(* IEC 61131-3 sources: Nauka-PLC-ST/, 81 files *)

(* ---- Zaawansowany_sterownik_prasy_hydraulicznej.st ---- *)
VAR
  stanAktualny               : stanPrasy;
  Przycisk_1                 : BOOL;  // pierwszy reczny przycisk uruchamiajacy prace ukladu
  Przycisk_2                 : BOOL;  // drugi reczny przycisk uruchamiajacy prace ukladu
  Dolna_krancowka_silownika  : BOOL;  // przelacznik krancowy wykrywajacy wysuniecie silownika
  Gorna_krancowka_silownika  : BOOL;  // przelacznik krancowy wykrywajacy wsuniecie silownika
  Timer_prasowanie           : TON;   // czas prasowania detalu
  Zawor_A                    : BOOL;  // zawor wysuwajacy prase w dol
  Zawor_B                    : BOOL;  // zawor wsuwajacy prase do gory
END_VAR

Timer_prasowanie(IN := Dolna_krancowka, PT := T#3S)

TYPE stanPrasy :
(
  OCZEKIWANIE
  RUCH_W_DOL
  PRASOWANIE
  RUCH_W_GORE
  ALARM
);
END_TYPE

CASE stanAktualny OF
    OCZEKIWANIE:
        Zawor_A := FALSE;
        Zawor_B := TRUE; // prasa czeka w górze

        // Warunek startu: Oba przyciski
        IF Przycisk_1 AND Przycisk_2 THEN
            stanAktualny := RUCH_W_DOL;
        END_IF;

    RUCH_W_DOL:
        Zawor_A := TRUE;  // Jedziemy w dół
        Zawor_B := FALSE;

        // oczekiwanie na stan wysoki od dolnej krancowki
        IF Dolna_krancowka_silownika THEN
            stanAktualny := PRASOWANIE;
        END_IF;

    PRASOWANIE:
        // wlaczamy timer (IN := TRUE)
        Timer_prasowanie(IN := TRUE, PT := T#3S);

        IF Timer_prasowanie.Q THEN
            Timer_prasowanie(IN := FALSE); // reset timera przed powrotem
            stanAktualny := RUCH_W_GORE;
        END_IF;

    RUCH_W_GORE:
        Zawor_A := FALSE;
        Zawor_B := TRUE; // powrot prasy do stanu poczatkowego

        IF Gorna_krancowka_silownika THEN
            stanAktualny := OCZEKIWANIE;
        END_IF;

    ALARM:
        Zawor_A := FALSE;
        Zawor_B := FALSE; // sytuacja awaryjna
END_CASE

(* ---- Motor_Control_Diagnostic.st ---- *)
FUNCTION_BLOCK Motor_control_diagnostic
VAR_INPUT
    xStart    : BOOL; // Przycisk Start
    xStop     : BOOL; // Przycisk Stop
    xFeedback : BOOL; // Potwierdzenie, ze silnik faktycznie ruszyl
    xErrorIn  : BOOL; // Awaria zewnetrzna (np. termik)
    xReset    : BOOL; // Przycisk do kasowania bledu
END_VAR

VAR_OUTPUT
    xRun      : BOOL;   // Wyjscie na stycznik silnika
    xAlarm    : BOOL;   // Lampka alarmu
    sStatus   : STRING; // Tekstowy opis na ekran HMI
END_VAR

VAR
    Timer_Potw : TON; // Zegar/czasowka
END_VAR

// --- 1. LOGIKA START / STOP ---
// Silnik rusza, gdy wciskasz Start, pod warunkiem, ze nie ma awarii i alarmu
IF xStart AND NOT xErrorIn AND NOT xAlarm THEN
    xRun := TRUE;
    sStatus := 'Silnik pracuje';
END_IF;

// Silnik staje, gdy: wcisniesz Stop, wywali blad (ErrorIn) lub pojawi sie Alarm
IF xStop OR xErrorIn OR xAlarm THEN
    xRun := FALSE;
    // Jesli to nie byl alarm, ustaw status na postoj
    IF NOT xAlarm THEN
        sStatus := 'Postoj';
    END_IF;
END_IF;

// --- 2. CZASOWKA (DIAGNOSTYKA) ---
// Timer liczy, gdy: wykonuje sie praca (xRun), ale nie widzisz potwierdzenia (NOT xFeedback)
Timer_Potw(IN := (xRun AND NOT xFeedback), PT := T#2s);

// --- 3. REAKCJA NA BLAD ---
// Jesli timer doliczyl do 2 sekund (Q), to znaczy, ze cos jest nie tak
IF Timer_Potw.Q THEN
    xAlarm  := TRUE;             // Wlaczamy alarm
    sStatus := 'Blad potwierdzenia'; // Opisujemy blad
    xRun    := FALSE;            // Wylaczamy silnik dla bezpieczenstwa
END_IF;

// --- 4. KASOWANIE ALARMU ---
// Gdy operator wcisnie Reset, czyscimy alarm i status
IF xReset THEN
    xAlarm := FALSE;
    sStatus := 'Gotowy';
END_IF;

(* ---- Obsluga_alarmow_analogowych.st ---- *)
FUNCTION_BLOCK Obsluga_alarmow_analogowych

VAR_INPUT
    Wartosc_Skalowana : REAL;    // Wartosc przeliczona
    Prog_Wysoki       : REAL;    // Prog alarmu
    Prog_Krytyczny    : REAL;    // Prog krytycznej wartosci w ukladzie
    Histereza         : REAL := 1.0; // Zapobiega przeciwko tzw drganiu stykow
END_VAR

VAR_OUTPUT
    Ostrzezenie : BOOL; // Informacja o przekroczeniu progu wysokiego
    Alarm       : BOOL; // Informacja o przekroczeniu progu krytycznego
END_VAR

// 1. Sprawdzenie progu krytycznego - natychmiastowe zatrzymanie, gdy zostanie przekroczona wartosc krytyczna
IF Wartosc_Skalowana >= Prog_Krytyczny THEN
    Alarm := TRUE;  // Informacja o przekroczeniu progu krytycznego
ELSIF Wartosc_Skalowana <= (Prog_Krytyczny - Histereza) THEN  // Wylacz alarm po powrocie do bezpiecznej wartosci
    Alarm := FALSE;  // Wylacz alarm
END_IF;

// 2. Ostrzezenie - tylko sygnalizacja
IF Wartosc_Skalowana >= Prog_Wysoki THEN
    Ostrzezenie := TRUE;  // Sygnalizacja przekroczenia normy np. lampka
ELSIF Wartosc_Skalowana <= (Prog_Wysoki - Histereza) THEN // Wylacz jesli spadnie ponizej tego progu
    Ostrzezenie := FALSE;
END_IF;

(* ---- Skalowanie_Analogowe.st ---- *)
FUNCTION_BLOCK Skalowanie_Analogow
VAR_INPUT
    Sygnal_RAW      : INT;    // Faktyczny odczyt z karty
    Zakres_Wej_Min   : REAL := 0.0;
    Zakres_Wej_Max   : REAL := 27648.0;
    Limit_Dolny     : REAL := 0.0;     // np. 0 bar
    Limit_Gorny     : REAL := 100.0;   // np. 10 bar
END_VAR

VAR_OUTPUT
    Wynik_Skalowania : REAL;    // Wartość przeliczona
    Awaria_Czujnika  : BOOL;    // Błąd zakresu / przerwany przewod
END_VAR

VAR
    Pomoc_Real       : REAL;    // Przejście na wartosc przecinkowa
END_VAR

// 1. Przepisanie wartosci z czujnika na wartosc z przecinkiem
Pomoc_Real := INT_TO_REAL(Sygnal_RAW);

// 2. Skalowanie wartosci z czujnika na wartosci fizyczne
IF (Zakres_Wej_Max - Zakres_Wej_Min) <> 0 THEN
    Wynik_Skalowania := Limit_Dolny + (Pomoc_Real - Zakres_Wej_Min) * (Limit_Gorny - Limit_Dolny) / (Zakres_Wej_Max - Zakres_Wej_Min);
ELSE
    Wynik_Skalowania := 0.0;
    Awaria_Czujnika := TRUE;
END_IF;

// 3. Diagnostyka na wypadek awarii
IF Pomoc_Real < -500.0 OR Pomoc_Real > 30000.0 THEN
    Awaria_Czujnika := TRUE;
ELSE
    Awaria_Czujnika := FALSE;
END_IF;

(* ---- Automat_segregujacy.st ---- *)
VAR
    Krok : INT := 0;              // krok programu
    Start_Maszyny : BOOL;         // przycisk NO wlaczajacy maszyne
    E_Stop : BOOL;                // przycisk bezpieczeństwa NC

    Tasma : BOOL;                 // napęd taśmociągu
    Spychacz_Metal : BOOL;        // aiłownik zrzucający metal
    Spychacz_Plastik : BOOL;      // aiłownik zrzucający plastik

    Fotokomorka_wlotowa : BOOL;   // wykrycie obiektu na wejściu
    Czujnik_indukcyjny : BOOL;    // detekcja metalu
    Czujnik_pojemnosciowy : BOOL; // detekcja plastiku
    Krancowka_baza : BOOL;        // czujnik potwierdzajacy powrotu siłowników na pozycję startowa

    Timer_Dojazdu : TON;          // Odmierzenie drogi od czujnika do spychacza
END_VAR

// system bezpieczenstwa
IF NOT E_stop THEN
    Tasma := FALSE;
    Spychacz_metal := FALSE;
    Spychacz_plastik := FALSE;
    Krok := 0;
    RETURN;
END_IF;

Timer_Dojazdu(IN := (Krok = 20 OR Krok = 30), PT := T#3s);

CASE Krok OF
    0:  // IDLE: oczekiwanie na gotowosc systemu
        Tasma := FALSE;
        IF Start_maszyny THEN
            Krok := 10;
        END_IF;

    10: // taśma rusza i czeka na materiał
        Tasma := TRUE;
        IF Czujnik_indukcyjny THEN
            Krok := 20; // wykrycie metalu
        ELSIF Czujnik_pojemnosciowy THEN
            Krok := 30; // wykrycie plastiku
        END_IF;

    20: // transportowaie metalu do spychacza
        IF Timer_dojazdu.Q THEN
            Tasma := FALSE;
            Krok := 21;
        END_IF;

    21: // uzycie silownika
        Spychacz_metal := TRUE;
        IF NOT Krancowka_baza THEN  // wysuniety spychacz
            Krok := 22;
        END_IF;

    22: // powrot spychacza do bazy
        Spychacz_metal := FALSE;
        IF Krancowka_baza THEN
            Krok := 10; // oczekiwanie na kolejen smieci
        END_IF;

    30: // transport plastiku
        IF Timer_dojazdu.Q THEN
            Tasma := FALSE;
            Krok := 31;
        END_IF;

    31: // zrzut plastiku do pojemnika
        Spychacz_plastik := TRUE;
        IF NOT Krancowka_baza THEN
            Krok := 32;
        END_IF;

    32: // powrot do stanu wyjsciowego
        Spychacz_plastik := FALSE;
        IF Krancowka_baza THEN
            Krok := 10;
        END_IF;

END_CASE;

(* ---- Automatyczny_cykl_nawrotny.st ---- *)
VAR
    Stycznik_lewo  : BOOL;
    Stycznik_prawo : BOOL;
    Przycisk_start : BOOL;
    Przycisk_stop  : BOOL; // Zakladamy NC

    Timer_pracy    : TON;
    Timer_pauzy    : TON;

    Kierunek       : BOOL; // FALSE = Lewo, TRUE = Prawo
    Praca_aktywna  : BOOL; // Informuje o uruchomionym cyklu
END_VAR

// Start i Stop cyklu
IF Przycisk_start AND Przycisk_stop THEN
    Praca_aktywna := TRUE;
ELSIF NOT Przycisk_stop THEN
    Praca_aktywna := FALSE;
END_IF;

// Obsluga timerow
Timer_pracy(IN := Praca_aktywna AND NOT Timer_pauzy.IN, PT := T#5S);
Timer_pauzy(IN := Timer_pracy.Q, PT := T#3S); // Czas na wyhamowanie

// Zmiana kierunku po kazdej pauzie
IF Timer_pauzy.Q THEN
    Kierunek := NOT Kierunek; // Przelacz na przeciwny
END_IF;

// Kontrola stycznikow
Stycznik_lewo  := Praca_aktywna AND NOT Kierunek AND NOT Timer_pauzy.IN;
Stycznik_prawo := Praca_aktywna AND Kierunek AND NOT Timer_pauzy.IN;

(* ---- Automatyczny_mieszalnik.st ---- *)
// 1. Obsługa Stopu Awaryjnego (Reset wszystkiego)
IF NOT Stop_awaryjny THEN
    Krok_ukladu := 0;
    Zawor_A := FALSE;
    Zawor_B := FALSE;
    Mieszadlo := FALSE;
    Zawor_spustowy := FALSE;
END_IF;

// 2. Główna maszyna stanów
CASE Krok_ukladu OF
    0: // Oczekiwanie
        IF Start THEN
            Krok_ukladu := 10;
        END_IF;

    10: // Dolewanie A
        Zawor_A := TRUE;
        IF Czujnik_poziomu >= 40.0 THEN
            Zawor_A := FALSE; // Wyłączamy, gdy pełne!
            Krok_ukladu := 20;
        END_IF;

    20: // Dolewanie B
        Zawor_B := TRUE;
        IF Czujnik_poziomu >= 80.0 THEN // Używaj tej samej nazwy zmiennej poziomu
            Zawor_B := FALSE;
            Krok_ukladu := 30;
        END_IF;

    30: // Mieszanie
        Mieszadlo := TRUE;
        // Składnia timera: Czas_mieszania(IN := TRUE, PT := T#10S);
        IF Czas_mieszania.Q THEN
            Mieszadlo := FALSE;
            Krok_ukladu := 40;
        END_IF;

    40: // Opróżnianie
        Zawor_spustowy := TRUE;
        IF Czujnik_poziomu <= 2.0 THEN
            Zawor_spustowy := FALSE;
            Krok_ukladu := 0; // Koniec cyklu, wróć do początku
        END_IF;
END_CASE;

(* ---- Diagnostyka_uszkodzenia_czujnika.st ---- *)
VAR
  wartoscCzujnik : REAL;  // wartosc odczytana z czujnika
  ostatniaWartosc : REAL;  // ostatnia wartosc z czujnika
  timerKontrola : TON;  // czas sprawdzania wartosci zmiany
  bladCzujnika : BOOL;  // pamiec bledu
  tolercjaSygnalu : REAL := 0.01;  // minimalna mozliwa zmiana aby program ja zauwazyl
END_VAR

// sprawdzenie odleglosci miedzy dwiema liczbami
IF ABS(wartoscCzujnik - ostatniaWartosc) < tolercjaSygnalu THEN
    // gdy tolerancja miedzy sygnalami jest za mala to uruchom odliczanie
    timerKontrola.IN := TRUE;
ELSE
    // gdy jednak sygnal sie zmienia to zresetuj timer
    timerKontrola.IN := FALSE;
END_IF;

timerKontrola.PT := T#10s; // deadline ze czujnik jest uszkodzony
timerKontrola();           // wywolanie timera kontroli sygnalu

IF timerKontrola.Q THEN
    bladCzujnika := TRUE;  // sygnalizacja alarmu
END_IF;

ostatniaWartosc := wartoscCzujnik;  // zapamietanie ostatniej wartosci czujnika

(* ---- Emergency_Stop.st ---- *)
PROGRAM SafetyLogic
VAR
    // WEJŚCIA
    bEStop_NC    : BOOL;    // Przycisk bezpieczeństwa (Fizycznie NC - Normalnie Zamknięty)
    bReset_Button : BOOL;   // Przycisk Reset (NO)

    // WYJŚCIA
    bSafetyOK    : BOOL;    // Flaga bezpieczeństwa - zezwolenie na pracę
    bError_Lamp  : BOOL;    // Lampa błędu (miga, gdy brak bezpieczeństwa)
END_VAR

// 1. Logika bezpieczeństwa
// Jeśli grzyb jest wciśnięty (bEStop_NC = FALSE), bezpieczeństwo zostaje przerwane
IF NOT bEStop_NC THEN
    bSafetyOK := FALSE;
END_IF

// 2. Warunek Resetu
// Bezpieczeństwo można przywrócić tylko, gdy grzyb jest wyciągnięty (TRUE)
// i naciśniemy przycisk Reset
IF bEStop_NC AND bReset_Button THEN
    bSafetyOK := TRUE;
END_IF

// 3. Sygnalizacja
bError_Lamp := NOT bSafetyOK;

END_PROGRAM

(* ---- Inteligentny_garaz.st ---- *)
VAR
    Wylacznik_ukladu    : BOOL;  // przcycisk bistabilny NC wylaczajacy brame
    Pilot_bramy         : BOOL;  // przycisk monostabilny NO otwierajacy brame
    Czujnik_ruchu_1     : BOOL;  // czujnik ruchu nr 1 w okolicach bramy
    Czujnik_ruchu_2     : BOOL;  // czujnik ruchu nr 2 w okolicach bramy
    Przycisk_serwisowy  : BOOL;  // przycisk NO monostabilny wlaczajacy swiatło na stałe
    Czujnik_CO2         : BOOL;  // czujnik wykrywajacy CO2 w powietrzu
    Potwierdzenie_went  : BOOL;  // potwierdzenie pracy wentylatora

    // --- WYJŚCIA (Fizyczne) ---
    Silnik_bramy        : BOOL;  // umozliwia wjazd samochodu
    Oswietlenie_bramy   : BOOL;  // oswietlenie bramy garazowej
    Wentylator          : BOOL;  // urzadzenie z podtrzymaniem
    Alarm_CO2           : BOOL; // czerwona lampka
    Alarm_Awaria_Went   : BOOL; // bład wentylatora/awaria wentylatora

    // --- BLOKI CZASOWE ---
    Timer_swiatlo       : TOF; // podtrzymanie światla po ruchu
    Timer_wentylator    : TOF; // podtrzymuje wietrzenie po zniknieciu gazu
    Timer_awaria_went   : TON; // odliczanie czasu na potwierdzenie pracy
END_VAR

// swiatlo reaguje na ruch, pdtrzymuje 30s po zniknieciu ruchu
Timer_swiatlo(IN := (Czujnik_ruchu_1 OR Czujnik_ruchu_2), PT := T#30s);

// wentylacja reaguje na gaz, trzyma 10s po oczyszczeniu powietrza
Timer_wentylator(IN := Czujnik_CO2, PT := T#10s);

// diagnostyka jeśli wentylator ma pracowac, a nie ma potwierdzenia przez 5s, a musi byc potwierdzenie
Timer_awaria_went(IN := Wentylator AND NOT Potwierdzenie_went, PT := T#5s);

// brama otwiera się z pilota, o ile nie ma gazu i system jest wlaczony
Silnik_bramy := Pilot_bramy AND NOT Czujnik_CO2 AND Wylacznik_ukladu;

// swiatlo: swieci gdy jest ruch (z podtrzymaniem), serwis, lub gdy brama pracuje
Oswietlenie_bramy := (Timer_swiatlo.Q OR Przycisk_serwisowy OR Silnik_bramy) AND Wylacznik_ukladu;

// wentylator pracuje na podstawie timera gazu
Wentylator := Timer_wentylator.Q AND Wylacznik_ukladu;

// alarmy
Alarm_CO2 := Czujnik_CO2;
Alarm_awaria_went := Timer_awaria_went.Q;

(* ---- Inteligentny_Sterownik_HVAC.st ---- *)
VAR
    Czujnik_hala    : REAL;    // czujnik glowny
    Hala_zapasowa   : REAL;    // czujnik zapasowy
    Wentylator      : BOOL;    // sterowanie silnikiem
    Alarm_czujnika  : BOOL;    // lampka awarii dowolnego czujnika
    Awaria_glowna   : BOOL;    // blad czujnika 1
    Awaria_zapas    : BOOL;    // blad czujnika 2
    Prog_temp       : REAL := 25.0; // prog zalaczenia wentylatora
    Blokada_systemu : BOOL;    // blad obu czujnikow
END_VAR

// Kontrola ciaglosci kabli
Awaria_glowna := (Czujnik_hala < -50.0) OR (Czujnik_hala > 150.0);
Awaria_zapas  := (Hala_zapasowa < -50.0) OR (Hala_zapasowa > 150.0);

// Alarm dziala gdy chociaz jeden czujnik ulegnie uszkodzeniu
Alarm_czujnika := Awaria_glowna OR Awaria_zapas;

// Jesli glowny czujnik sie zepsuje to system patrzy na zapasowy
IF NOT Awaria_glowna THEN
    // Uzycie glownego czujnika
    IF Czujnik_hala > Prog_temp THEN
        Wentylator := TRUE;
    ELSIF Czujnik_hala < (Prog_temp - 2.0) THEN
        Wentylator := FALSE;
    END_IF;

ELSIF Awaria_glowna AND NOT Awaria_zapas THEN
    // Awaria - uzywanie zapasowego czujnika
    IF Hala_zapasowa > Prog_temp THEN
        Wentylator := TRUE;
    ELSIF Hala_zapasowa < (Prog_temp - 2.0) THEN
        Wentylator := FALSE;
    END_IF;

ELSE
    // Oba czujniki ulegly uszkodzeniu
    Blokada_systemu := TRUE;
    Wentylator := TRUE; // Uruchamiamy chlodzenie
END_IF;

// wylaczenie blokady jesli chociaz jeden czujnik wroci do pracy
IF NOT Awaria_glowna OR NOT Awaria_zapas THEN
    Blokada_systemu := FALSE;
END_IF;

(* ---- Kontrola_przepelnienia_bufora.st ---- *)
VAR
    Fotokomorka_bufora   : BOOL;  // czujnik optyczny na koncu
    Podajnik_glowny_On   : BOOL;  // sygnal ze glowny podajnik podaje paczki

    Timer_przepelnienia  : TON;   // timer mierzacy czas pelnego zasloniecia czujnika
    Licznik_zatrzyman    : CTU;   // licznik rejestrujacy ilosc awaryjnych zatrzyman

    Zatrzymanie_awaryjne : BOOL;  // blokada zatrzymujaca glowny podajnik
END_VAR

// Badanie czasu zaslonietego czujnika przez conajmniej 4 sekundy - bufor jest pelny
Timer_przepelnienia(IN := Fotokomorka_bufora AND Podajnik_glowny_On, PT := T#4s);

// 2.Logika blokady
Zatrzymanie_awaryjne := Timer_przepelnienia.Q;

// Tworzenie statystyki - licznik zwieksza swoja wartosc gdy bufor sie przepelni
Licznik_zatrzyman(CU := Timer_przepelnienia.Q, R := NOT Podajnik_glowny_On);

(* ---- Kontrola_ruchu_rasmy.st ---- *)
(* Potwierdzenie ruchu poprzez czujnik obrotów *)

VAR
    OpoznienieStartu      : TON;    // Czas na rozbieg
    TimeoutBrakuRuchu     : TON;    // Czas oczekiwania na kolejny impuls
    WykrywanieObrotow     : R_TRIG; // Detekcja sygnału z czujnika
    CzujnikWykrywajacyRuch : BOOL;   // Potwierdzenie obrotu taśmy
END_VAR

// 1. Dajemy maszynie czas na ruszenie
OpoznienieStartu(IN := Silnik_Praca, PT := T#3S);

// 2. Wykrycie impulsu ruchu
WykrywanieObrotow(CLK := Sygnal_z_czujnika);

// 3. Kontrola alarmów przy pracy
IF Silnik_Praca AND OpoznienieStartu.Q THEN

    // Wykrycie obrotu - taśma pracuje poprawnie
    IF WykrywanieObrotow.Q THEN
        TimeoutBrakuRuchu(IN := FALSE);
        CzujnikWykrywajacyRuch := TRUE;
    ELSE
        // Brak impulsu - odliczanie czasu do błędu
        TimeoutBrakuRuchu(IN := TRUE, PT := T#800MS);
    END_IF;

ELSE
    TimeoutBrakuRuchu(IN := FALSE);
    CzujnikWykrywajacyRuch := FALSE;
END_IF;

// 4. Reakcja na błąd
IF TimeoutBrakuRuchu.Q THEN
    WykrycieBleduRuchu := TRUE;
    Silnik_Praca := FALSE; // Zatrzymanie silnika po przekroczeniu czasu timeout
END_IF;

(* ---- Kontrola_wentylatora.st ---- *)
VAR
    Start_przycisk : BOOL;
    Stop : BOOL;            // Zakładamy styk NC (TRUE = OK, FALSE = STOP)
    Potwierdzenie : BOOL;   // Sygnał z czujnika przepływu
    Wentylator : BOOL;
    Alarm : BOOL;
    Flaga_awarii : BOOL;
    Temperatura_aktualna : REAL;

    Timer_rozbieg : TON;    // Czas na rozpędzenie
    Timer_awarii : TON;     // Czas na wykrycie braku przepływu
END_VAR

// Obsługa Timerów (muszą być wywoływane co cykl)
Timer_rozbieg(IN := Wentylator, PT := T#5S);
// Timer awarii startuje tylko gdy wentylator już się rozpędził, a przepływu brak
Timer_awarii(IN := Timer_rozbieg.Q AND NOT Potwierdzenie, PT := T#2S);

// Start układu
IF Start_przycisk AND Stop AND NOT Flaga_awarii THEN
    Wentylator := TRUE;
END_IF;

// Wyłączenie przez przycisk STOP lub awarię
IF NOT Stop OR Flaga_awarii THEN
    Wentylator := FALSE;
END_IF;

// Detekcja awarii (Brak przepływu LUB za wysoka temperatura)
IF Timer_awarii.Q OR (Wentylator AND Temperatura_aktualna > 80.0) THEN
    Flaga_awarii := TRUE;
    Alarm := TRUE;
END_IF;

// Reset awarii (Przyciskiem Stop)
IF NOT Stop AND Flaga_awarii THEN
    Flaga_awarii := FALSE;
    Alarm := FALSE;
END_IF;

(* ---- Licznik_godzin_pracy.st ---- *)
(* Licznik czasu pracy napedu *)

VAR
    TaktSekundowy       : TON;    // Odmierzanie kazdej sekundy pracy
    SumaSekund          : DINT;   // Skumulowany czas pracy [s]
    GodzinyPracy        : REAL;   // Czas pracy wyswietlany na HMI [h]
    Limit_Przegladu     : REAL := 500.0; // Czas do wezwania serwisu [h]
    PrzypomnienieSerwisu: BOOL;   // Aktywacja przypomnienia o przegladzie
    Reset_Serwisu       : BOOL;   // Potwierdzenie wykonania prac serwisowych
END_VAR

// 1. Odmierzanie czasu tylko podczas pracy silnika
TaktSekundowy(IN := Silnik_Praca AND NOT TaktSekundowy.Q, PT := T#1S);

// 2. Zliczanie czasu i przeliczanie na godziny
IF TaktSekundowy.Q THEN
    SumaSekund := SumaSekund + 1;

    // Przeliczenie sekund na godziny (1h = 3600s)
    GodzinyPracy := DINT_TO_REAL(SumaSekund) / 3600.0;
END_IF;

// 3. Sprawdzenie czy nadszedl czas na serwis
IF GodzinyPracy >= Limit_Przegladu THEN
    PrzypomnienieSerwisu := TRUE;
END_IF;

// 4. Kasowanie licznika po wykonaniu serwisu
IF Reset_Serwisu THEN
    SumaSekund := 0;
    PrzypomnienieSerwisu := FALSE;
END_IF;

(* ---- Licznik_godzin_z_blokada.st ---- *)
VAR
    Timer_1s : TON;              // timer zliczajacy ilosc sekund pracy silnika
    Silnik : BOOL;               // stycznik silnika
    Reset_serwis : BOOL;         // przycisk serwisowy
    Sygnalizacja_serwisu : BOOL; // lampa serwisowa
    Licznik_serwisu : DINT;      // tu przechowujemy sekundy
END_VAR

// odmierzanie kazdej sekundy
Timer_1s( IN := Silnik AND NOT Timer_1s.Q, PT := T#1s);

// suma czasu
IF Timer_1s.Q THEN
    Licznik_serwisu := Licznik_serwisu + 1;
END_IF;

// sprawdzaie czasu serwisowego
IF Licznik_serwisu >= 32400 THEN
    Sygnalizacja_serwisu := TRUE;
    Silnik := FALSE; // Blokada silnika
ELSE
    Silnik := TRUE;  // Pozwolenie na pracę, jeśli serwis nie jest wymagany
END_IF;

// reset czasu serwisu
IF Reset_serwis THEN
    Sygnalizacja_serwisu := FALSE;
    Licznik_serwisu := 0;
END_IF;

(* ---- Licznik_paczek.st ---- *)
VAR
    Numer_stanowiska : INT;      // wybor jednego stanowiska z pieciu
    Dodaj_paczke : BOOL;         // sygnal z czujnika/przycisku
    Reset_total : BOOL;          // zerowanie licznikow

    // Definicja tablicy
    Licznik_paczki : ARRAY[0..4] OF INT; // tablica przechowujaca wyniki

    i : INT;                     // licznik do petli FOR
    R_Trig_Paczka : R_TRIG;      // wykrywanie zbocza
END_VAR

// detekcja zbocza
R_Trig_Paczka(CLK := Dodaj_paczke);

// dodawanie paczki z kontrola zakresu
IF R_Trig_Paczka.Q AND (Numer_stanowiska >= 0 AND Numer_stanowiska <= 4) THEN
    // zwiekszamy wartosc w wybranej "szufladce"
    Licznik_paczki[Numer_stanowiska] := Licznik_paczki[Numer_stanowiska] + 1;
END_IF;

// czyszczenie wszystkich stanowisk (Reset)
IF Reset_total THEN
    // petla FOR przechodzi przez 0, 1, 2, 3, 4
    FOR i := 0 TO 4 DO
        Licznik_paczki[i] := 0;
    END_FOR;
END_IF;

(* ---- Licznik_wydajnosci_z_rejestrem.st ---- *)
VAR
    Ostatnie_czasy : ARRAY[1..5] OF TIME;  // tablica z czasami
    Indeks_zapisu : INT := 1;  // wskaznik mowiacy do jakiej komorki tablicy zapisac czas
    Sensor_wyjscie : BOOL;  // czujnik wykrywajacy fizyczny przejazd pudelka
    Aktualny_czas_pudelka : TIME;   // zmienna czasowa jak dlugo pudelko bylo pakowane
    Sredni_czas : TIME;  // zmienna do wyniku obliczen z pakowania 5 ostatnich pudelek
    Suma_czasow : LINT;  // zamianana typu TIME na  i sumowanie czasow w tej komorce
    i : INT;  // licznik petli
    Trigger_Sensor : R_TRIG;  // zbocze narastajace
END_VAR

// wykrycie zbocza (impulsu) czujnika
Trigger_Sensor(CLK := Sensor_wyjscie);

IF Trigger_Sensor.Q THEN
    // zapis do tablicy
    Ostatnie_czasy[Indeks_zapisu] := Aktualny_czas_pudelka;

    // przesunięcie indeksu
    Indeks_zapisu := Indeks_zapisu + 1;

    // po zapelnieniu calej talicy wracamy na poczatek
    IF Indeks_zapisu > 5 THEN
        Indeks_zapisu := 1;
    END_IF;
END_IF;

// obliczanie sredniej i sumowanie wyniku
Suma_czasow := 0;

FOR i := 1 TO 5 DO
    // sumowanie wszystkich elementów tablicy
    Suma_czasow := Suma_czasow + TIME_TO_LINT(Ostatnie_czasy[i]);
END_FOR;

// wynik sredniej czasu
Sredni_czas := LINT_TO_TIME(Suma_czasow / 5);

(* ---- Logika_tasmociagu.st ---- *)
VAR
    Start_linii      : BOOL;   // przycisk Start (NO)
    Bit_pracy_linii  : BOOL;   // bit pracy linii
    Stop_linii       : BOOL;   // przycisk Stop (NC)
    Czujnik_obecnosci: BOOL;   // fotokomorka na końcu tasmy
    Reset_alarmu     : BOOL;   // przycisk potwierdzenia awarii
    Silnik_tasmy     : BOOL;   // wyjście na stycznik silnika
    Alarm_zator      : BOOL;   // czerwona lampka alarmowa
    Timer_eco        : TOF;    // timer podtrzymujący bieg tasmy
    Timer_zator      : TON;    // timer wykrywajacy blokade
END_VAR

Timer_eco(IN := Start_linii OR Czujnik_obecnosci, PT := T#10s);  // wlaczamy zegar przyciskiem start, kazda paczka resetuje czas i liczy ponowne 10 s
Timer_zator(IN := Czujnik_obecnosci, PT := T#5s);

IF Start_linii AND Stop_linii AND NOT Alarm_zator THEN  // aktywacja gotowej linii bez awarii  //
  Bit_pracy_linii := TRUE;  // uruchomienie pracy linii
END_IF;

IF Timer_eco.Q AND NOT Czujnik_obecnosci AND NOT Stop_linii THEN  // wylaczenie pracy po czasie bezczynnosci bez paczek
  Silnik_tasmy := 0;
  Bit_pracy_linii := FALSE;
END_IF;

IF Timer_zator.Q THEN  // aktwyacja alarmu gdy czujnik wykrywa obiekt zbyt dlugo
  Silnik_tasmy := FALSE;
  Alarm_zator := TRUE;
END_IF;

IF Timer_zator.Q AND NOT Czujnik_obecnosci AND Reset_alarmu THEN
  Alarm_zator := FALSE;
END_IF;

Silnik_tasmy := Bit_pracy_linii AND Timer_eco.Q AND NOT Alarm_zator;  // sterowanie napedem z uzglednieniem trybu eco oraz blokady startu

(* ---- Lube_control.st ---- *)
VAR
    Wlacznik_Start      : BOOL;   // Przycisk monostabilny NO (Start)
    Przycisk_Stop       : BOOL;   // Przycisk monostabilny NC (Stop)
    Reset_alarmu        : BOOL;   // Przycisk kasowania błędów
    Cisnienie_smaru     : REAL;   // Wartość ciśnienia w układzie [bar]

    Silnik_hala         : BOOL;   // Stycznik silnika głównego
    Pompa_smaru         : BOOL;   // Wyjście sterujące pompą smaru

    Maszyna_Pracuje     : BOOL;   // Flaga stanu pracy (Zatrzask SET/RESET)
    Licznik_cyklu       : INT;    // Ilość cykli pracy maszyny
    Alarm_ukladu        : BOOL;   // Pamięć błędu krytycznego
    Status_maszyny      : STRING; // Informacja tekstowa dla operatora
    Reset_Timera        : BOOL;   // Sygnał odświeżenia timera 8h

    Czas_pracy          : TON;    // Odlicza 8h do kolejnego smarowania
    Timer_cisnienia     : TON;    // Czeka 30s na nabicie ciśnienia
    R_Trig_Puls         : R_TRIG; // Wykrywa moment startu silnika
END_VAR

// maszyna rusza po wicsnieciu start jesli nie ma alarmu
IF Wlacznik_Start AND NOT Alarm_ukladu THEN
    Maszyna_Pracuje := TRUE;
END_IF;

// zatrzymmanie maszyny po stop lub alarmie ukladu
IF Przycisk_Stop OR Alarm_ukladu THEN
    Maszyna_Pracuje := FALSE;
END_IF;

// czas pracy gdy maszyna pracuje, nie liczy sie czas smarowania
Czas_pracy(IN := Maszyna_Pracuje AND NOT Pompa_smaru AND NOT Reset_Timera, PT := T#8h);

// cykliczny czas smarowania
Timer_cisnienia(IN := Pompa_smaru, PT := T#30s);

// zliczanie ilosci uruchomien maszyny
R_Trig_Puls(CLK := Maszyna_Pracuje);

IF R_Trig_Puls.Q THEN
    Licznik_cyklu := Licznik_cyklu + 1;
END_IF;

// cykliczne smarowanie pompy po 8h lub 100 cyklach
IF Czas_pracy.Q OR Licznik_cyklu >= 100 THEN
    Pompa_smaru := TRUE;
END_IF;

// wylaczenie pompy po osiagnieciu cisnienia
IF Pompa_smaru AND Cisnienie_smaru >= 50.0 THEN
    Pompa_smaru    := FALSE;
    Licznik_cyklu  := 0;
    Reset_Timera   := TRUE;  // Puls resetujący timer TON
ELSE
    Reset_Timera   := FALSE;
END_IF;

// alarm gdy po 30 sekundach pracy pompy nie ma cisnienia
IF Timer_cisnienia.Q AND Cisnienie_smaru < 50.0 THEN
    Alarm_ukladu := TRUE;
    Pompa_smaru  := FALSE; // Ochrona pompy przed pracą na sucho
END_IF;

// kasowanie alarmu
IF Reset_alarmu THEN
    Alarm_ukladu := FALSE;
END_IF;

// statusy
IF Alarm_ukladu THEN
    Status_maszyny := 'Awaria: ZA NISKIE CISNIENIE SMARU';
ELSIF Pompa_smaru THEN
    Status_maszyny := 'TRWA SMAROWANIE...';
ELSIF Maszyna_Pracuje THEN
    Status_maszyny := 'PRACA NORMALNA';
ELSE
    Status_maszyny := 'MASZYNA ZATRZYMANA';
END_IF;

// sterowanie stycznikiem glownego napedu
Silnik_hala := Maszyna_Pracuje;

(* ---- Monitor_wydajnosci_cyklu.st ---- *)
VAR
    Stoper_Cyklu     : TON;         // timer mirzacy czas trwania cyklu
    Czas_Ostatni     : TIME;        // ostatni zapisany wynik
    Limit_Czasu      : TIME := T#10S; // limit do uruchomienia alarmu
    Alarm_Wydajnosci : BOOL;
END_VAR

// 1. Logika stopera - działa gdy prasa NIE JEST w stanie OCZEKIWANIE ani ALARM
// mierzenie czasu od startu ruchu w dół do powrotu na górę
Stoper_Cyklu(IN := (stanAktualny <> OCZEKIWANIE AND stanAktualny <> ALARM), PT := T#60S);

// zbocze gdy maszyna wrocila do stanu poczatkowego
IF stanAktualny = OCZEKIWANIE AND Stoper_Cyklu.ET > T#0S THEN
    Czas_Ostatni := Stoper_Cyklu.ET; // aktualnie liczony czas timera ET
END_IF;

// detekcja czy maszyna nie pracuje za wolno
Alarm_Wydajnosci := Czas_Ostatni > Limit_Czasu;

(* ---- Monitoring_obciazenia_silnika.st ---- *)
VAR
    Przycisk_start : BOOL;         // przycisk NO monostabilny uruchamiajacy uklad
    Przycisk_stop : BOOL;          // przycisk NC bistabilny wylaczajacy uklad
    Potwierdzenie_awarii : BOOL;   // przycsik NO monostabilny potwierdzajacy awarie
    Prad_silnika : INT;            // miernik pradu na silniku wartosc 0-1000
    Temp_uzwojenia : INT;          // czujnik temperatur yan silniku wartosc 0-150
    Stycznik_silnika : BOOL;       // stycznik zasilajacy silnik
    Lamp_ostrzezenie : BOOL;       // lampa sygnalizujaca przeciazenie silnika
    Syrena_przeciazenia : BOOL;    // sygnal dzwiekowy informujacy o przeciazeniu
    Blokada_Awaryjna : BOOL;       // flaga pamietajaca wystapienie awarii
    Timer_przeciazenia : TON;      // czas opoznienia stanu przeciazenia silnika
    Licznik_uruchomien : CTU;      // ilosc uruchomien silnika
END_VAR

// deklaracja timera
Timer_przeciazenia(IN := (Prad_silnika >= 900), PT := T#5S);

// licznik uruchomien silnika
Licznik_uruchomien(CU := Stycznik_silnika);

// wykrycie awarii i blokada silnika
IF Timer_przeciazenia.Q OR Temp_uzwojenia > 110 THEN
    Blokada_Awaryjna := TRUE;   // aktywacja flagii awarii
    Stycznik_silnika := FALSE;  // natychmiastowe wyłączenie silnika
    Syrena_przeciazenia := TRUE;  // wlaczenie syerny ifnormujacej o przeciazeniu
END_IF;

// ostrzezenie, silnik jeszcze pracuje
IF Prad_silnika > 700 THEN
    Lamp_ostrzezenie := TRUE;
ELSE
    Lamp_ostrzezenie := FALSE;
END_IF;

// reset awarii gdy silnik ostygl i zostal wcisniety przycisk
IF Potwierdzenie_awarii AND Temp_uzwojenia < 60 THEN
    Blokada_Awaryjna := FALSE;
    Syrena_przeciazenia := FALSE;
END_IF;

// sterowanie silnikiem gdy nie ma blokady
IF Przycisk_start AND NOT Blokada_Awaryjna AND Przycisk_stop THEN
    Stycznik_silnika := TRUE;
END_IF;

IF NOT Przycisk_Stop THEN  // wcisniecie przycisku lub zerwanie kabla wylacza silnik
    Stycznik_silnika := FALSE;
END_IF;

(* ---- Myjnia_samochodowa.st ---- *)
VAR
    Przycisk_start : BOOL;  // przycisk monostabilny NO wlaczajacy uklad
    Przycisk_stop : BOOL;   // przycisk monostabilny NC zatrzymujacy prace ukladu
    Szczotki_naped : BOOL;  // silniki szczotek czyszczacych auto
    Wentylator_suszarka : BOOL;  // wyjscie wentylatora suszacego samochod
    Zawor_woda : BOOL;  // zawor wody do mycia i splukiwania
    Zawor_szampon : BOOL;  // zawor podajacy szampon samochodowy

    // deklaracja wszystkich timerow dla kazdego kroku
    Czas_kroku_1 : TON;  // czas namaczania
    Czas_kroku_2 : TON;  // czas mcyai zasadniczego
    Czas_kroku_3 : TON;  // czas plukania
    Czas_kroku_4 : TON;  // czas suszenia

    Stan : INT := 0; // aktualny krok
END_VAR

// logika timerow
// timery mierza czas gdy dany stan jest aktywny
Czas_kroku_1(IN := (Stan = 1), PT := T#5S);  // czas namaczania
Czas_kroku_2(IN := (Stan = 2), PT := T#10S); // czas mycia zasadniczego
Czas_kroku_3(IN := (Stan = 3), PT := T#5S);  // czas plukania
Czas_kroku_4(IN := (Stan = 4), PT := T#8S);  // czas suszenia

// zatrzymanie o najwiekszym priorytecie
IF NOT Przycisk_stop THEN // jesli  wcisniety grzyb NC = FALSE to alarm
    Stan := 0;
    Zawor_woda := 0;
    Zawor_szampon := 0;
    Szczotki_naped := 0;
    Wentylator_suszarka := 0;
END_IF;

// kroki myjni

// #1 namaczanie
IF Przycisk_start AND Przycisk_stop AND Stan = 0 THEN  // namaczanie samochodu
    Stan := 1;
    Zawor_woda := 1;
END_IF;

// #2: mycie zasadnicze
IF Czas_kroku_1.Q AND Stan = 1 THEN
    Stan := 2;
    Zawor_woda := 1;
    Szczotki_naped := 1;
    Zawor_szampon := 1;
END_IF;

// #3: plukanie
IF Czas_kroku_2.Q AND Stan = 2 THEN
    Stan := 3;
    Szczotki_naped := 0;
    Zawor_szampon := 0;
    Zawor_woda := 1;
END_IF;

// #4: suszenie
IF Czas_kroku_3.Q AND Stan = 3 THEN
    Stan := 4;
    Zawor_woda := 0;
    Wentylator_suszarka := 1; // Uruchomienie nadmuchu
END_IF;

// koniec cyklu
IF Czas_kroku_4.Q AND Stan = 4 THEN
    Stan := 0; // powrot do oczekiwania na sygnal
    Wentylator_suszarka := 0; // wylaczenie suszenia
END_IF;

(* ---- Nawadnianie_ogrodu.st ---- *)
VAR
    Czujnik_deszczu : BOOL;         // TRUE = pada deszcz
    Wilgotnosc_gleby : INT;        // 0-100% wilgotnosci
    Zawór_wody : BOOL;              // wyjscie na elektrozawór

    Zegar : RTC;                    // czas systemowy
    Godzina : INT;

    Timer_podlewania : TON;         // czas pracy zraszaczy
    Krok : INT := 0;                // Maszyna stanów
END_VAR

VAR_CONSTANT
    Prog_wilgotnosci : INT := 40;   // podlewaj tylko ponizej 40% wilgotnosci
    Czas_podlewania : TIME := T#15M; // czas trwania podlewania
    Godzina_startu : INT := 5;      // start o 5:00 rano
END_VAR

// zmienne zegara
Zegar();
Godzina := Zegar.CDT.Hour;

// czas podlewania
Timer_podlewania(IN := (Krok = 2), PT := Czas_podlewania);

CASE Krok OF
    0: // czekanie na podlewanie
        Zawór_wody := FALSE;
        IF Godzina = Godzina_startu THEN
            Krok := 1;
        END_IF;

    1: // analizowanie warunków pogodowych
        IF NOT Czujnik_deszczu AND (Wilgotnosc_gleby < Prog_wilgotnosci) THEN
            Krok := 2; // podlej gdy jest sucho
        ELSE
            Krok := 3; // omin podlewanie gdy jest mokro
        END_IF;

    2: // podlewanie
        Zawór_wody := TRUE;
        IF Timer_podlewania.Q THEN
            Krok := 3;
        END_IF;

    3: // Blokada po cyklu (czekamy, az minie godzina startu)
        Zawór_wody := FALSE;
        IF Godzina <> Godzina_startu THEN
            Krok := 0; // powrot do stanu poczatkowego gdy nastanie odpowiednia godzina
        END_IF;
END_CASE;

(* ---- Oświetlenie_korytarzowe.st ---- *)
VAR
    Czujnik_ruchu : BOOL;                   // czujnik wykrywajacy ruch, ruch = TRUE
    Czujnik_natezezenia_oswietlenia : INT;  // fotokomorka w [luks]
    Zegar_systemowy : RTC;                  // blok zegara czasu rzeczywistego
    Aktualna_godzina : INT;                 // faktyczna godzina (liczba)

    Modul_sciemniajacy : INT;               // wartosc 0-100% mocy lamp
    Krok : INT := 0;                        // krok ukladu sekwencyjnego

    Timer_brak_ruchu : TON;                 // oczekiwanie przy braku ruchu
    Timer_wylaczenia : TON;                 // czas calkowitego wylaczenia ze standby
END_VAR

VAR_CONSTANT
    Moc_dzien : INT := 100;                 // moc oswietlenia w dzien
    Moc_noc : INT := 30;                    // moc oswietlenia w noc
    Moc_standby : INT := 10;                // oswietlenie gdy na korytarzu nikogo nie ma
    Prog_lux : INT := 500;                  // powyzej tej wartosci uklad nie swieci
END_VAR

// dane w programie
Zegar_systemowy();
Aktualna_godzina := Zegar_systemowy.CDT.Hour; // Pobranie aktualnej godziny do obliczeń

// czas przejscia systemu w standby (30 sekund braku ruchu)
Timer_brak_ruchu(IN := NOT Czujnik_ruchu, PT := T#30S);

// po 5 minutach w kroku standby oswietlenie wylaczy sie calkowicie
Timer_wylaczenia(IN := (Krok = 2), PT := T#5M);

// logika programu
CASE Krok OF

    0: // wylaczenie - oszczedzanie energii
        Modul_sciemniajacy := 0;

        // wykrycie ruchu w korytarzu gdy jest ciemno
        IF Czujnik_ruchu AND (Czujnik_natezezenia_oswietlenia < Prog_lux) THEN
            Krok := 1;
        END_IF;

    1: // oswietlenie dostosowane do pory dnia
        // Sprawdzenie godziny: dzien (6-22) czy noc
        IF (Aktualna_godzina >= 6 AND Aktualna_godzina < 22) THEN
            Modul_sciemniajacy := Moc_dzien; // Pełna moc 100%
        ELSE
            Modul_sciemniajacy := Moc_noc;   // Moc zredukowana 30%
        END_IF;

        // brak ruchu przez 30 s - sciemnij do standby
        IF Timer_brak_ruchu.Q THEN
            Krok := 2;
        END_IF;

    2: // standby czuwanie - 10% mocy
        Modul_sciemniajacy := Moc_standby;

        // wykryty ruch - powrot do pelnego swiatla (Krok 1)
        IF Czujnik_ruchu THEN
            Krok := 1;
        END_IF;

        // wylaczenie ukladu po 5 minutach bez ruchu lub gdy zrobi sie widno
        IF Timer_wylaczenia.Q OR (Czujnik_natezezenia_oswietlenia > Prog_lux) THEN
            Krok := 0;
        END_IF;

END_CASE;

(* ---- Prasa_hydrauliczna.st ---- *)
// aby prasa dzialala trzeba wcisnac przycisk_1 i przycisk_2

VAR
    Przycisk_1        : BOOL; // przycisk uruchamiajacy lewy
    Przycisk_2        : BOOL; // przycisk uruchamiajacy prawy
    Praca             : INT := 0;  // Krok ukladu: 0-Oczekiwanie na wlaczenie, 1-silownik w dol, 2-postoj silownika, 3-silownik w gore
    Zawor_wysun       : BOOL;
    Zawor_schowaj     : BOOL;
    Liczba_sztuk      : INT := 0;
    Czujnik_swietlny  : BOOL;  // czujnik bezpieczenstwa NC
    Timer_postoju     : TON;
END_VAR

// przecieta wiazka z czujnika swietlnego - powrot silownikow
IF NOT Czujnik_swietlny AND (Praca = 1 OR Praca = 2) THEN
    Praca := 3;
END_IF;

// maszyna stanow
CASE Praca OF

    0: // OCZEKIWANIE NA URUCHOMIENIE
        Zawor_wysun   := FALSE;
        Zawor_schowaj := TRUE;
        IF Przycisk_1 AND Przycisk_2 AND Czujnik_swietlny THEN
            Praca := 1;
        END_IF;

    1: // SILOWNIK W DOL
        Zawor_wysun   := TRUE;
        Zawor_schowaj := FALSE;
        // Tutaj w realu byłby czujnik krańcowy, ale załóżmy, że dojechał:
        IF Przycisk_1 AND Przycisk_2 THEN // przejscie do kolejnego kroku jesli przyciski stan wysoki
             Praca := 2;
        ELSIF NOT (Przycisk_1 AND Przycisk_2) THEN  // puszczenie przycisku przed zakonczenie pracy
             Praca := 3;
        END_IF;

    2: // OCZEKIWANIE I DOCISK SILOWNIKA 3 sekundy
        Timer_postoju(IN := TRUE, PT := T#3s);
        IF Timer_postoju.Q THEN
            Liczba_sztuk := Liczba_sztuk + 1; // ziczenie dodatkowej sztuki
            Timer_postoju(IN := FALSE);      // reset timera
            Praca := 3;
        END_IF;

    3: // POWRÓT DO GÓRY
        Zawor_wysun   := FALSE;
        Zawor_schowaj := TRUE;
        //wroc do kroku zero po powrocie silownika
        Praca := 0;

END_CASE;

(* ---- Production_counter.st ---- *)
PROGRAM ProductionCounter
VAR
    // --- WEJŚCIA CYFROWE ---
    bSensor_PartDetected : BOOL;    // Sygnał z fotokomórki (TRUE = detal wykryty)
    bReset_Counter       : BOOL;    // Fizyczny przycisk zerowania licznika

    // --- PARAMETRY I USTAWIENIA ---
    iTarget_Quantity    : INT := 10; // Docelowa liczba detali w jednym opakowaniu

    // --- PAMIĘĆ WEWNĘTRZNA ---
    bSensor_LastState    : BOOL;    // Przechowuje stan czujnika z poprzedniego cyklu sterownika

    // --- WYJŚCIA I STATUSY ---
    iCurrent_Count      : INT := 0;  // Suma zliczonych detali w aktualnej partii
    bBox_Full           : BOOL;      // Sygnał zakończenia pakowania (osiągnięto limit)
END_VAR

// 1. Logika wykrywania zbocza narastającego (R_TRIG - zobacze narastające)
// Sprawdzamy czy teraz jest sygnał, a w poprzednim cyklu go nie było. Zapobiega to wielokrotnemu zliczaniu tego samego detalu.
IF bSensor_PartDetected AND NOT bSensor_LastState THEN
    iCurrent_Count := iCurrent_Count + 1; // Inkrementacja licznika
END_IF
// Przepisujemy aktualny stan na "stary", aby użyć go w następnym obiegu pętli
bSensor_LastState := bSensor_PartDetected;

// 2. Kontrola wypełnienia (Porównanie)
// Jeśli licznik osiągnie lub przekroczy limit, wystawiamy sygnał pełnego kartonu.
IF iCurrent_Count >= iTarget_Quantity THEN
    bBox_Full := TRUE;  // Aktywacja wyjścia
ELSE
    bBox_Full := FALSE; // Wyłączenie sygnału, jeśli licznik jest poniżej limitu
END_IF

// 3. Obsługa zerowania systemu
// Jeśli operator naciśnie przycisk Reset, licznik wraca do zera.
IF bReset_Counter THEN
    iCurrent_Count := 0; // Zerowanie wartości aktualnej
END_IF

END_PROGRAM

(* ---- Przeszukiwanie _tablicy.st ---- *)
VAR
    // tablica z danymi - 5 wartosci
    Licznik_Paczki : ARRAY[0..4] OF INT := [12, 45, 7, 23, 10];

    // zmienne
    Max_Wartosc : INT;      // Ile paczek ma lider
    Lider_Stanowisko : INT; // Numer stanowiska-lidera

    // zmienne pomocnicze
    i : INT;                // Licznik do pętli
END_VAR

//poszukiwanie najwiekszej wartosci
Max_Wartosc := 0; // czyszczenie przed kazdym szukanie

FOR i := 0 TO 4 DO
    // wartosc wieksza niz dotychzawsowy max
    IF Licznik_Paczki[i] > Max_Wartosc THEN
        // wybranie najwieskzej wartosci
        Max_Wartosc := Licznik_Paczki[i];
        Lider_Stanowisko := i; // zapamietaj numer komorki
    END_IF;
END_FOR;

(* ---- Regulacja_poziomu_w_zbiorniku_z_histereza.st ---- *)
(* Regulacja poziomu w zbiorniku z histereza miedzy 20 a 80 procent zapelnienia w zbiorniku *)

VAR
    Poziom_aktualny  : REAL;    // Odczyt z czujnika faktycznego poziomu wody w zbiorniku [0.0 - 100.0 %]
    Prog_niski       : REAL := 20.0;
    Prog_wysoki      : REAL := 80.0;

    Pompa_dolewowa   : BOOL;    // Obsluga stycznika pompy
    Blad_czujnika    : BOOL;    // Zmienna awarii
END_VAR

// 1. Detekcja awarii czujnika (wartosci niemozliwe)
IF Poziom_aktualny < -5.0 OR Poziom_Aktualny > 105.0 THEN
    Blad_czujnika := TRUE;
ELSE
    Blad_czujnika := FALSE;
END_IF;

// 2. Logika regulacji
IF Blad_czujnika THEN
    Pompa_dolewowa := FALSE; // Bezpieczeństwo: stop przy awarii

ELSIF Poziom_aktualny <= Prog_niski THEN
    Pompa_dolewowa := TRUE;  // Startuje pompe dopiero na samym dole (20%)

ELSIF Poziom_aktualny >= Prog_wysoki THEN
    Pompa_dolewowa := FALSE; // Wyłączam pompe dopiero przy pelnym zbiorniku (80%)

END_IF;

(* ---- Rotacja_Pracy_Pomp.st ---- *)
VAR
    niskiPoziomWody   : BOOL; // wykrycie niskiego poziomu wody w zbiorniku
    kolejPompy1       : BOOL := TRUE; // pamiec ktora pompa ma dzialac
    zboczeNiskiPoziom : R_TRIG; // zbocze wykrywajace niski poziom

    Pompa_1           : BOOL; // stycznik sterujacy pompa #1
    Pompa_2           : BOOL; // stycznik sterujacy pompa #2
END_VAR

// wkrycie niskiego poziomu wody w zbiorniku
zboczeNiskiPoziom(CLK := niskiPoziomWody);

// wykryto zbocze, zmien priorytet pomp
IF zboczeNiskiPoziom.Q THEN
    kolejPompy1 := NOT kolejPompy1;
END_IF;

// sterowanie pompami - pompa pracuje gdy jest niski poziom wody oraz jest jej kolej do pracy
Pompa_1 := niskiPoziomWody AND kolejPompy1;
Pompa_2 := niskiPoziomWody AND NOT kolejPompy1;

(* ---- Sekwencyjne_wlaczanie_silnikow.st ---- *)
(* Rozruch kaskadowy linii tasmociagow *)

VAR
    Przycisk_Start   : BOOL;    // Przycisk Start (NO)
    Przycisk_Stop    : BOOL;    // Przycisk Stop (NC)
    System_Aktywny   : BOOL;    // Flaga pamieci ukladu

    Zwloka_S2        : TON;     // Czas oczekiwania na silnik 2
    Zwloka_S3        : TON;     // Czas oczekiwania na silnik 3

    Silnik_1         : BOOL;
    Silnik_2         : BOOL;
    Silnik_3         : BOOL;
END_VAR

// 1. Logika zalaczania ukladu - podtrzymanie
IF Przycisk_Start AND Przycisk_Stop THEN
    System_Aktywny := TRUE;
ELSIF NOT Przycisk_Stop THEN
    System_Aktywny := FALSE;
END_IF;

// 2. Uklad kaskadowy - kazdy kolejny krok wynika z poprzedniego
Silnik_1 := System_Aktywny;

Zwloka_S2(IN := Silnik_1, PT := T#5S);
Silnik_2 := Zwloka_S2.Q;

Zwloka_S3(IN := Silnik_2, PT := T#5S);
Silnik_3 := Zwloka_S3.Q;

(* ---- Sekwencyjny_rozruch_wentylatorow.st ---- *)
VAR
    Start_wentylacji     : BOOL;  // przycisk uruchomienia systemu wentylacji
    Stop_wentylacji      : BOOL;  // przycisk wylaczenia calego ukladu

    Timer_rozruchu       : TON;   // timer odmierzajacy czas pomiedzy startami kolejnych silnikow
    Etap                 : INT;   // aktualny krok sekwencji rozruchu: 0-stop, 1-went1, 2-went2, 3-went3
    System_aktywny       : BOOL;  // flaga pamieciowa pracy systemu (zatrzask)

    Wentylator_1         : BOOL;  // cewka stycznika pierwszego wentylatora
    Wentylator_2         : BOOL;  // cewka stycznika drugiego wentylatora
    Wentylator_3         : BOOL;  // cewka stycznika trzeciego wentylatora
END_VAR

// start/stop
IF Start_wentylacji THEN
    System_aktywny := TRUE;
ELSIF Stop_wentylacji THEN
    System_aktywny := FALSE;
    Etap           := 0; // reset sekwencji rozruchu
END_IF;

// logika sekwencji
IF System_aktywny THEN
    CASE Etap OF
        0: // Krok 0: uruchomienie pierwszego wentylatora
            Etap := 1;

        1: // czas na rozpedzenie obydwu wentylatorow
            IF Timer_rozruchu.Q THEN
                Etap := 2;
            END_IF;

        2: // oczekwianie na rozpedzenie wentylatorow
            IF Timer_rozruchu.Q THEN
                Etap := 3;
            END_IF;

        3: // wszystkie prawidlowo pracujace wentylatory - koniec sekwencji
    END_CASE;
END_IF;

// rozruch - zwloka 5 sekund
// Timer odlicza czas w krokach przejsciowych (1 oraz 2), dajac czas na rozped silnikow
Timer_rozruchu(IN := (Etap = 1) OR (Etap = 2), PT := T#5s);

// sterowanie wyjsciami
Wentylator_1 := System_aktywny AND (Etap >= 1);
Wentylator_2 := System_aktywny AND (Etap >= 2);
Wentylator_3 := System_aktywny AND (Etap >= 3);

(* ---- Skalowanie_analogowe.st ---- *)
VAR
    // wejścia wyjścia
    raw_Input : INT;          // sygnał z czujnika 0-32767
    scaled_value : REAL;      // wynik w jednostkach w bar

    // zmienne pomocnicze
    in_real : REAL;           // konwersja wartosci wejsciowej

    // alarmy
    alarm_HH : BOOL;          // alarm - za wysokie cisnienie
    alarm_LL : BOOL;          // alarm - za niskie cisnienie
END_VAR

VAR_CONSTANT
    Raw_Max : REAL := 32767.0; // maksymalna wartosc plc
    EU_Max : REAL := 10.0;     // maksymalne cisnienie
    limit_HH : REAL := 9.5;    // wartosc alarmu wysokiego
    limit_LL : REAL := 0.5;    // wartosc alarmu nisokiego
END_VAR

// konwersja danych
in_real := INT_TO_REAL(raw_input);

// skalowanie
// obliczamy jaki to procent zakresu i mnożymy przez wartość maksymalną
scaled_value := (in_real / raw_max) * EU_Max;

// kontrola limitow
// kontrola niskiego cisnienia
IF scaled_value >= limit_HH THEN
    alarm_HH := TRUE;
ELSE
    alarm_HH := FALSE;
END_IF;

// Sprawdzanie niskiego ciśnienia
IF scaled_value <= limit_LL THEN
    alarm_LL := TRUE;
ELSE
    alarm_LL := FALSE;
END_IF;

(* ---- Skalowanie_analogowe_PT100.st ---- *)
VAR
    Raw_Input : INT;          // bezposrednia wartość z wejścia analogowego
    Temp_Min : REAL := -50.0; // Dolny sygnal czujnika
    Temp_Max : REAL := 150.0; // Górny sygnal czujnika
    Current_Temp : REAL;      // Obliczona temperatura w stopniach C
    Alarm_Przegrzania : BOOL; // Sygnał alarmowy
END_VAR

// 1. Skalowanie - zamiana INT na REAL ze wzrou
// uzycie instrukcji INT_TO_REAL
Current_Temp := (INT_TO_REAL(Raw_Input) / 27648.0) * (Temp_Max - Temp_Min) + Temp_Min;

// 2. Instrukcja alarmu
IF Current_Temp > 100.0 THEN
    Alarm_Przegrzania := TRUE;
ELSE
    Alarm_Przegrzania := FALSE; // wyłączenie alarmu gdy temp. spadnie!
END_IF;

(* ---- Skalowanie_poziomu_w_zbiorniku.st ---- *)
VAR
    Surowe_wejscie : INT;      // wartosc z czujnika
    Wejscie_Real   : REAL;     // zmienna
    Poziom_metry   : REAL;     // wartosc w zbiorniku
    Alarm_wysoki   : BOOL;
END_VAR

// 1. Konwersja INT na REAL (dzielenie z przecinkiem)
Wejscie_Real := INT_TO_REAL(wartosc z konwersja na real);

Poziom_metry := (Wejscie_Real / 27648.0) * 10.0;  // zasosowanie zrobu do czujnika

// zabezpieczenie aby wartosc nie byla ujemna
IF Poziom_metry > 10.0 THEN
    Poziom_metry := 10.0;
ELSIF Poziom_metry < 0.0 THEN
    Poziom_metry := 0.0;
END_IF;

// alarm
IF Poziom_metry > 9.0 THEN
    Alarm_wysoki := TRUE;
ELSIF Poziom_metry < 8.5 THEN
    Alarm_wysoki := FALSE;
END_IF;

(* ---- Sortowanie_gabarytow_tasmy.st ---- *)
VAR
    Fotokomorka_pomiaru   : BOOL;  // czujnik optyczny PNP wykrywajacy paczke
    Tasma_praca           : BOOL;  // potwierdzenie ze tasmociag sie porusza

    Timer_gabarytu        : TON;   // timer mierzacy czas przykrycia fotokomorki
    Impuls_spychacza      : TOF;   // timer generujacy odpowiedni czas pracy silownika spychajacego

    Silownik_spychacza    : BOOL;  // wyjscie: sterowanie elektrozaworem siłownika spychajacego
    Licznik_gabarytow     : CTU;   // licznik zliczajacy odrzucone duze paczki
END_VAR

// Mierzenie czasu przejscia paczki
// Timer zaczyna odliczac czas, gdy paczka zasloni czujnik, pod warunkiem ze tasma jedzie. Gdy paczka zasloni czujnik na dluzej niz 1.5 sekundy to jest za duzy gabaryt
Timer_gabarytu(IN := Fotokomorka_pomiaru AND Tasma_praca, PT := T#1s500ms);

// Sterowanie silownikiem
// Gdy timer wykryje gabaryt generujemy impuls trwajacy 1 sekunde(wysuniecie silownika na boczny tor)
Impuls_spychacza(IN := Timer_gabarytu.Q, PT := T#1s);
Silownik_spychacza := Impuls_spychacza.Q;

// Statystyka
// Licznik zwieksza wartosc po kazdym wykrytym i odrzuconej paczce
Licznik_gabarytow(CU := Timer_gabarytu.Q, R := NOT Tasma_praca);

(* ---- Stacja_napelniania_butelek.st ---- *)
VAR
    fotokomorka : BOOL;   // wykrywa butelke
    waga : INT;           // odczyt wagi
    transporter : BOOL;    // silnik linii
    zawor : BOOL;         // zawor cieczy
    alarm : BOOL;         // alarm
    krok : INT := 0;      // krok ukladu
    czas_stabilizacji : TON; // deklaracja timera
END_VAR

VAR_CONSTANT
    wartosc_docelowa : INT := 500;
    tolerancja : INT := 5;
END_VAR

// wywołanie timera
czas_stabilizacji(IN := (krok = 3), PT := T#2S);

CASE krok OF
    0:  // oczekiwanie
alarm := FALSE;
transporter := TRUE;
        zawor := FALSE;
        IF fotokomorka THEN
            krok := 1;
        END_IF;

    1:  // Zatrzymanie i start nalewania
        transporter := FALSE;
        zawor := TRUE;
        krok := 2; // od razu do monitorowania wagi

    2:  // nalewanie cieczy
        IF waga >= wartosc_docelowa THEN
            zawor := FALSE;
            krok := 3;
        END_IF;

    3:  // stabilizacja
        IF czas_stabilizacji.Q THEN
            krok := 4;
        END_IF;

    4:  // Kontrola jakosci
        IF waga >= (wartosc_docelowa - tolerancja) AND
           waga <= (wartosc_docelowa + tolerancja) THEN
            krok := 0; // waga ok - następna butelka
        ELSE
            alarm := TRUE; // blad - stop
        END_IF;
END_CASE;

(* ---- Stacja_pakujaca.st ---- *)
VAR
    // WEJŚCIA
    Czujnik_paczki       : BOOL; // Czujnik wykrywający paczki (NO)
    Stop_awaryjny_NC     : BOOL; // Przycisk awaryjny (NC - True gdy jest OK)
    Silownik_wrocil      : BOOL; // Czujnik krańcowy pozycji bazowej siłownika

    // WYJŚCIA
    Silnik_tasmy         : BOOL; // Napęd taśmociągu
    Silownik_zrzutu      : BOOL; // Wyjście na siłownik spychający

    // BLOKI FUNKCYJNE
    Licznik_paczek       : CTU;  // Blok zliczający
    Timer_zrzutu         : TP;   // Generator impulsu 2s dla siłownika

    // USTAWIENIA
    Limit_paczek         : INT := 6;
END_VAR

// Licznik paczek - licznik zwiększa się, gdy paczka przetnie czujnik, nastapi reset gdy zruci paczki do pakowania
Licznik_paczek(CU := Czujnik_paczki,
               R := (Timer_zrzutu.Q = FALSE AND Licznik_paczek.Q),
               PV := Limit_paczek);

// Gdy licznik zrzuci paczki to zacznie jest zrzucac, bedzie to trwalo 2 sekundy
Timer_zrzutu(IN := Licznik_paczek.Q, PT := T#2s);

// Sterowanie silnikiem od tasmy - tasma caly czas jedzie dopoki nie ma stopu, pelnego kartonu
Silnik_tasmy := Stop_awaryjny_NC AND NOT Licznik_paczek.Q AND NOT Timer_zrzutu.Q;

// Sterowanie silownikiem pakujacym paczki - gdy chce pakowac to trwa to mu dwie sekundy
Silownik_zrzutu := Timer_zrzutu.Q AND Stop_awaryjny_NC;

(* ---- Stacja_sortujaca.st ---- *)
VAR
    Czujnik_paczki : BOOL;  // wykrycie produktu
    Waga_analogowa : INT;   // masa produktu wartosc 0-1000
    Przycisk_Reset : BOOL;  // resetowanie alarmu i licznikow
    Tasmociag : BOOL;       // silnik linii
    Silownik_odrzutu : BOOL;  // spychacz
    Lampa_Alarm : BOOL;     // sygnalizacja bledu
    Stan : INT := 0;        // krok maszyny

    Timer_Wazenia : TON;    // czas na zwazenie produktu
    Timer_Odrzutu : TON;    // czas wysuniecia silownika
    Timer_Dojazdu : TON;    // DODANO: czas przejazdu miedzy sekcjami

    Sztuki_OK : INT := 0;   // produkty poprawne
    Sztuki_NOK : INT := 0;  // produkty odrzucone
    Bledy_pod_rzad : INT := 0; //licznik bledow
    Alarm_Aktywny : BOOL := FALSE;
END_VAR

CASE Stan OF
0:  // --- Stan oczekiwania na sygnal ---
    Tasmociag := FALSE; // tasma stoi

    IF Czujnik_paczki AND NOT Alarm_Aktywny THEN
        Stan := 10;
    END_IF;

10: // --- Transport paczek ---
    Tasmociag := TRUE;

    // Paczka jedzie 3 sekundy pod wage
    Timer_Dojazdu(IN := TRUE, PT := T#3S);

    IF Timer_Dojazdu.Q THEN
        Timer_Dojazdu(IN := FALSE); // reset timera
        Tasmociag := FALSE;         // stop tasmy bo paczka jest na wadze
        Stan := 20;                 // nastepny krok - wazenie
    END_IF;

20: // wazenie paczki przez 2 sek
    Timer_Wazenia(IN := TRUE, PT := T#2S);

    IF Timer_Wazenia.Q THEN
        Timer_Wazenia(IN := FALSE); // reset timera wazenia

        // LOGIKA ANALIZY WAGI
        IF Waga_analogowa >= 400 AND Waga_analogowa <= 600 THEN
            // PACZKA POPRAWNA
            Sztuki_OK := Sztuki_OK + 1;
            Bledy_pod_rzad := 0; // wyzerowanie licznika bledow
            Stan := 30;          // przejscie do kolejnego kroku
        ELSE
            // PACZKA WADLIWA
            Sztuki_NOK := Sztuki_NOK + 1;
            Bledy_pod_rzad := Bledy_pod_rzad + 1; // Zliczamy bledy pod rzad
            Stan := 40;          // kolejny kroku odrzut
        END_IF;
    END_IF;

30: // transport poprawnej paczki
    Tasmociag := TRUE;

    // czas zjazdu z wagi
    Timer_Dojazdu(IN := TRUE, PT := T#3S);

    IF Timer_Dojazdu.Q THEN
       Timer_Dojazdu(IN := FALSE);
       Tasmociag := FALSE;
       Stan := 0; // wyzerowanie ukladu do stanu poczatkowego
    END_IF;

40: // przygotowanie do odrzutu paczki
    Tasmociag := TRUE;

    // Spychacz jest 2 sekundy za waga
    Timer_Odrzutu(IN := TRUE, PT := T#2S);

    IF Timer_Odrzutu.Q THEN
        Timer_Odrzutu(IN := FALSE);
        Tasmociag := FALSE; // zatrzymanie tasmy aby zepchnac
        Stan := 45;
    END_IF;

45: // praca spychacza
    Silownik_odrzutu := TRUE;

    Timer_Odrzutu(IN := TRUE, PT := T#1S);

    IF Timer_Odrzutu.Q THEN
        Timer_Odrzutu(IN := FALSE);
        Silownik_odrzutu := FALSE; // schowanie tloka
        Stan := 0;
    END_IF;

END_CASE;

// alarm
IF Bledy_pod_rzad >= 3 THEN
    Alarm_Aktywny := TRUE;
    Lampa_Alarm := TRUE;
END_IF;

IF Przycisk_Reset THEN
    Alarm_Aktywny := FALSE;
    Lampa_Alarm := FALSE;
    Bledy_pod_rzad := 0;
    Stan := 0;
END_IF;

(* ---- Sterowanie_dynamiczne_rampy.st ---- *)
VAR
    rTargetBrightness  : REAL := 0.0;   // wartosc docelowa jasnosci lampy
    rActualInternal    : REAL := 0.0;   // biezacy poziom jasnosci
    rRampSpeed         : REAL := 0.5;   // szybkosc zmiany wartosci na raz - skok rampy

    iAnalogOut         : INT;  // wartosc wysylkana na wyjscie fizyczne
    iMaxRaw            : INT := 27648;  // rozdzielczosc przetwornika
END_VAR

// jesli roznica jest mniejsza niz krok to ustaw wartosc docelowa
IF ABS(rTargetBrightness - rActualInternal) < rRampSpeed THEN
    rActualInternal := rTargetBrightness;

ELSIF rActualInternal < rTargetBrightness THEN
    rActualInternal := rActualInternal + rRampSpeed;  // w kazdym cyklu dodajemy maly kawalek jasnosci

ELSIF rActualInternal > rTargetBrightness THEN  // sprawdzenie czy jasnosc nie jest za duza
    rActualInternal := rActualInternal - rRampSpeed;
END_IF;

iAnalogOut := REAL_TO_INT((rActualInternal / 100.0) * INT_TO_REAL(iMaxRaw));  // zamiana wartosci 0100 na zakres 0-1.0

IF iAnalogOut > iMaxRaw THEN  // sprawdza czy wynik sie nie znalazl poza dopuszczalne wartosci
    iAnalogOut := iMaxRaw;  // nie pozwol wyjsc powyzej 27648
ELSIF iAnalogOut < 0 THEN
    iAnalogOut := 0;  // nie pozwala na wyjscie na wartosci ujemne
END_IF;

(* ---- Sterowanie_kaskadowe_pomp.st ---- *)
VAR
    Poziom : REAL;           // Sygnał z czujnika (0-100%)
    Pompa_1 : BOOL;
    Pompa_2 : BOOL;

    Zamiana : BOOL;          // Pamiec do zmiany kolejności
    Cykl_Aktywny : BOOL;     // Zabezpieczenie zmiany trybu pracy
END_VAR

// 1. Gdy zbiornik jest pusty
IF Poziom < 5.0 AND NOT Cykl_Aktywny THEN
    Zamiana := NOT Zamiana;
    Cykl_Aktywny := TRUE; // Blokada
END_IF;

IF Poziom > 10.0 THEN
    Cykl_Aktywny := FALSE; // Reset blokady - gdy zaczyna nalewać
END_IF;

// 2. Sterowanie
IF NOT Zamiana THEN
    // Kolejność: P1 główna, P2 pomocnicza
    Pompa_1 := Poziom > 70.0;
    Pompa_2 := Poziom > 90.0;
ELSE
    // Kolejność: P2 główna, P1 pomocnicza
    Pompa_2 := Poziom > 70.0;
    Pompa_1 := Poziom > 90.0;
END_IF;

// 3. Wyłącznik bezpieczeństwa
IF Poziom < 30.0 THEN
    Pompa_1 := FALSE;
    Pompa_2 := FALSE;
END_IF;

(* ---- Sterowanie_przepompownia.st ---- *)
VAR
    Poziom_metry      : REAL;    // Poziom cieczy w zbiorniku
    Czujnik_cisnienia : BOOL;    // Kontrola cisnienia w rurociągu
    Pompa_wyjscie     : BOOL;    // Wyjscie sterujace pompa
    Alarm_suchobieg   : BOOL;    // Alarm pracy bez cisnienia
    Licznik_uruchomien: INT;     // Licznik cykli pracy
    Przycisk_reset    : BOOL;    // Wejscie kasujace błąd

    Timer_cisnienia   : TON;     // Blok czasowy
    R_Trig_Pompa      : R_TRIG;  // Wykrywacz zbocza narastającego
END_VAR

// 1. logika Start/Stop
IF Poziom_metry >= 8.0 THEN
    Pompa_wyjscie := TRUE;
ELSIF Poziom_metry <= 2.0 OR Alarm_suchobieg THEN
    Pompa_wyjscie := FALSE;
END_IF;

// 2. zliczanie uruchomień
R_Trig_Pompa(CLK := Pompa_wyjscie);
IF R_Trig_Pompa.Q THEN
    Licznik_uruchomien := Licznik_uruchomien + 1;
END_IF;

// kontrola suchobiegu (Jeśli pompa pracuje, a ciśnienia brak przez 3s)
Timer_cisnienia(IN := Pompa_wyjscie AND NOT Czujnik_cisnienia, PT := T#3S);

IF Timer_cisnienia.Q THEN
    Alarm_suchobieg := TRUE; // Zatrzaśnięcie błędu (Latch)
END_IF;

// reset alarmu
IF Przycisk_reset THEN
    Alarm_suchobieg := FALSE;
END_IF;

(* ---- Sterowanie_sekwencyjne_tasmociagiem.st ---- *)
// Sterowanie sekwencyjne taśmociągiem (Automat Stanów)
// Główna logika zarządzająca procesem transportu detali.
// Wykorzystuje strukturę CASE do separacji stanów pracy.

// 1. Zastosowałem numerację co 10 (0, 10...), aby umożliwić łatwą rozbudowę
//    sekwencji o dodatkowe stany bez konieczności potrzeby przenumerowywania kodu.
// 2. Stan 99 zarezerwowano dla trybu EMERGENCY (Awaria) - wysoka wartość
//    pozwala na szybką identyfikację błędu w systemie monitoringu.

VAR
    iState          : INT := 0;     // Numer aktualnego stanu maszyny
    sStatus_Message : STRING;       // Komunikat tekstowy dla panelu HMI
    bMotor_Run      : BOOL;         // Wyjście fizyczne: Silnik napędu
    bStart_Button   : BOOL;         // Wejście: Przycisk START (NO)
    bStop_Button    : BOOL;         // Wejście: Przycisk STOP (NC)
    bSafety_OK      : BOOL;         // Sygnał z przekaźnika bezpieczeństwa
    bSensor_Full    : BOOL;         // Wejście: Czujnik zajętości odbioru
    bReset_Button   : BOOL;         // Wejście: Przycisk Reset błędu
END_VAR

// LOGIKA STEROWANIA
CASE iState OF

    0: // STAN: IDLE - Oczekiwanie na inicjację procesu
        bMotor_Run := FALSE;
        sStatus_Message := 'System gotowy - Oczekiwanie na START';

        // Wciśnięty start i obwód bezpieczeństwa jest zamknięty
        IF bStart_Button AND bSafety_OK THEN
            iState := 10;
        END_IF

    10: // STAN: PRACA - Praca automatyczna taśmociągu
        bMotor_Run := TRUE;
        sStatus_Message := 'Produkcja w toku - Taśma pracuje';

        // Powrót jeśli naciśnięto STOP lub czujnik wykrył zator (pełny karton)
        IF bStop_Button OR bSensor_Full THEN
            iState := 0;
        END_IF

        // Priorytetowe przejście do stanu awaryjnego przy sygnale E-Stop
        IF NOT bSafety_OK THEN
            iState := 99;
        END_IF

    99: // STAN: EMERGENCY - Blokada po naruszeniu bezpieczeństwa
        bMotor_Run := FALSE; // Natychmiastowe zatrzymanie napędu
        sStatus_Message := 'ALARM: Naruszone bezpieczeństwo! Wymagany Reset';

        // Powrót do trybu gotowości tylko po przywróceniu bezpieczeństwa i potwierdzeniu
        IF bSafety_OK AND bReset_Button THEN
            iState := 0;
        END_IF

    ELSE // Zabezpieczenie przed nieoczekiwaną wartością iState program przechodzi w tryb czekania na sygnał
        iState := 0;

END_CASE

(* ---- Sterowanie_tasmy.st ---- *)
VAR
    // WEJŚCIA
    bStart      : BOOL;    // Przycisk Start (NO)
    bStop       : BOOL;    // Przycisk Stop (NC)

    // WYJŚCIA
    bSilnik     : BOOL;    // Stycznik silnika taśmy
    bLampa      : BOOL;    // Lampa sygnalizacyjna

    // WEWNĘTRZNE
    fbTimer     : TON;     // Timer do opóźnienia startu
    bPraca      : BOOL;    // Flaga stanu pracy
END_VAR

// 1. Logika Start/Stop (Podtrzymanie)
IF bStart AND bStop THEN
    bPraca := TRUE;
ELSIF NOT bStop THEN
    bPraca := FALSE;
END_IF

// Timer opóźniający start silnika (3 sekundy ostrzeżenia)
fbTimer(IN := bPraca, PT := T#3s);

// Sterowanie wyjściami
bSilnik := fbTimer.Q;      // Silnik rusza dopiero po odliczeniu czasu
bLampa  := bPraca AND NOT fbTimer.Q; // Lampa świeci tylko podczas odliczania timera

END_PROGRAM

(* ---- Sterownik_bramy_z_kurtyna.st ---- *)
VAR
    Krok : INT := 0;
    Listwa_optyczna : BOOL;    // Bezpieczeństwo (0 = przeszkoda / przerwana wiązka)
    Silnik_gora : BOOL;   // stycznik podnoszacy brame
    Silnik_dol : BOOL;   // stycznik opuszczajacy brame
    Krancowka_gora : BOOL;  // czujnik wykrwyajacy brame w gornej krancowej pozycji
    Krancowka_dol : BOOL;  // czujnik krancowy wykrywajacy brame w dolnej krancowej pozycji
    Petla_indukcyjna : BOOL;   // petla indukcyjna wykrwyajaca wozek widlowy
    Kurtyna_wyjscie : BOOL;    // uklad sterujacy kurtyna

    Licznik_cykli : INT;       // licznik zliczajacy ilosc wykonanej pracy ukladu
    Timer_kurtyny : TOF;       // czas dzialania ukladu po zamknieciu
    Odjazd_wozka : TON;        // czas oczekiwania ukladu na przejazd wozka
END_VAR

// timery - kurtyna dziala gdy brama sie rusza lub nie jest calkowicie zamknieta
Timer_kurtyny(IN := (Krok > 0), PT := T#10S);  // dalsza praca ukladu po wykonaniu pelnego cyklu
Kurtyna_wyjscie := Timer_kurtyny.Q;

// czas na przejazd wozka gdy brama jest w gorze
Odjazd_wozka(IN := (Krok = 2), PT := T#5S);

// maszyna stanow
CASE Krok OF
    0: // brama zamknięta
        Silnik_gora := FALSE;
        Silnik_dol := FALSE;

        IF Petla_indukcyjna THEN
            Licznik_cykli := Licznik_cykli + 1; // dodanie nowego cyklu pracy
            Krok := 1;
        END_IF;

    1: // otwieranie
        Silnik_gora := TRUE;

        IF Krancowka_gora THEN
            Silnik_gora := FALSE;
            Krok := 2;
        END_IF;

    2: // brama otwarta - oczekiwanie 5s aż wózek przejedzie
        IF Odjazd_wozka.Q THEN
            Krok := 3;
        END_IF;

    3: // zamykanie bramy
       // braca tylko gdy listwa optyczna nic nie wykryje
        IF NOT Listwa_optyczna THEN
            Silnik_dol := FALSE; // stop gdy listwa optyczna cos wykryje
            Krok := 1;  // gdy wykryje przeszkode brama w gore
        ELSE
            Silnik_dol := TRUE;
        END_IF;

        IF Krancowka_dol THEN
            Silnik_dol := FALSE;
            Krok := 0; // powrot do stanu poczatkowego - kurtyna i tak będzie działać przez TOF
        END_IF;

        // wykrycie wozka podczas zamykania - brama do gory
        IF Petla_indukcyjna THEN
            Silnik_dol := FALSE;
            Krok := 1;
        END_IF;
END_CASE;

(* ---- Sterownik_centrali_wentylacyjnej.st ---- *)
VAR
    Moj_czas_struktura : DTL;        // struktura siemensa zawierajaca rok, miesiac, godzine
    Status_funkcji     : INT;        // informacja diagnostyczna
    Godzina_system     : INT;        // pamiec dla pobranej godziny (od 0 do 23)
    Tryb_nocny         : BOOL;       // flaga: TRUE = jest noc (18-6), FALSE = jest dzień
    Sygnal_CO2_RAW     : INT;        // surowy sygnal z czujnika fizycznego (od 0 do 27648)
    Poziom_CO2         : REAL;       // przeliczona wartosc (0 - 2000 ppm)
    Wydajnosc_nawiew   : REAL;       // sygnal dla wentylatora: jak mocno ma dmuchac (0% - 100%)
END_VAR

Status_funkcji := RD_LOC_T(OUT => Moj_Czas_Struktura);
Godzina_system := Moj_czas_struktura.HOUR;

Tryb_nocny := (Godzina_system >= 18) OR (Godzina_system < 6);
Poziom_CO2 := (INT_TO_REAL(Sygnal_CO2_RAW) / 27648.0) * 2000.0;

// logika sterowania
IF Tryb_nocny THEN
    Wydajnosc_nawiew := 10.0;
ELSE
    // praca dzienna uzalezniona od ilosci CO2
    IF Poziom_CO2 > 1000.0 THEN  // duze stezenie CO2, bardzo wysokie --> mocne wietrzenie
        Wydajnosc_nawiew := 100.0;
    ELSIF Poziom_CO2 > 700.0 THEN   // podwyzszone stezenie CO2, zwiekszona wentylacja
        Wydajnosc_nawiew := 75.0;
    ELSE
        Wydajnosc_nawiew := 50.0;  // standardowy poziom CO2, normalna wentylacja
    END_IF;

END_IF;

(* ---- Sterownik_czyszczenia.st ---- *)
VAR
    Start_czyszczenia    : BOOL;  // przycisk uruchomienia procedury mycia CIP
    Potwierdzenie_pompy  : BOOL;  // sygnal zwrotny prawidlowo pracujacej pompy

    Timer_etapu          : TON;   // timer mierzacy faze mycia
    Etap                 : INT;   // krok ukladu sekwencyjnego

    Zawor_wody_surowej   : BOOL;  // cewka zaworu podajacego wode do plukania wstepnego
    Zawor_srodka_chem    : BOOL;  // cewka zaworu podajacego goracy roztwor myjacy
    Zawor_wody_czystej   : BOOL;  // cewka zaworu podajacego wode do plukania koncowego
    Pompa_obiegowa_CIP   : BOOL;  // cewka pompy obiegowej podajacej wode przez rurociagi
END_VAR

CASE Etap OF
    0: // uklad czekajacy na sygnal
        IF Start_czyszczenia THEN
            Etap := 1; // przejscie do plukania wstepnego
        END_IF;

    1: // plukanie wstepne woda surowa
        IF Timer_etapu.Q THEN
            Etap := 2; // przejscie do mycia zasadniczego
        END_IF;

    2: // mycie goracym srodkiem czyszczacym
        IF Timer_etapu.Q THEN
            Etap := 3; // przejscie do koncowego plukania
        END_IF;

    3: // plukanie na koniec czysta woda
        IF Timer_etapu.Q THEN
            Etap := 0; // koniec calej sekwencji, uklad wraca do oczekiwania na sygnal
        END_IF;
END_CASE;

// przypisanie czasu dla kazdej z faz mycia
IF Etap = 1 THEN
    Timer_etapu(IN := Potwierdzenie_pompy, PT := T#15s);
ELSIF Etap = 2 THEN
    Timer_etapu(IN := Potwierdzenie_pompy, PT := T#30s);
ELSIF Etap = 3 THEN
    Timer_etapu(IN := Potwierdzenie_pompy, PT := T#20s);
ELSE
    Timer_etapu(IN := FALSE);
END_IF;

// sterowanie wyjsciami
Zawor_wody_surowej := (Etap = 1); // cewka zaworu otwartego podczas plukania wstepnego
Zawor_srodka_chem  := (Etap = 2); // cewka zaworu otwartego podczas mycia chemia
Zawor_wody_czystej := (Etap = 3); // cewka zaworu otwartego podczas plukania koncowego
Pompa_obiegowa_CIP := (Etap > 0); // pompa pracujaca w kazdym etapie mycia

(* ---- Sterownik_czyszczenia_wymiennika.st ---- *)
VAR
    Temperatura_wlot     : REAL;  // temperatura spalin przed wymiennikiem
    Temperatura_wylot    : REAL;  // temperatura spalin za wymiennikiem
    Zgoda_na_przedmuch   : BOOL;  // cisnienie powietrza w zbiorniku jest prawidlowe

    Timer_sekcji         : TON;   // czas otwarcia zaworu danego obszaru podczas czyszczenia
    Krok                 : INT;   // krok sekwencji

    Sprawnosc_niska      : BOOL;  // zmienna informujaca o uruchomieniu cyklu
    Zawor_sekcji_1       : BOOL;  // zawor elektro-pneumatyczny sekcji pierwszej
    Zawor_sekcji_2       : BOOL;  // zawor elektro-pneumatyczny sekcji drugiej
END_VAR

// gdy roznica temperatur spadnie ponizej 15 stopni to wymiennik jest zabrudzony
IF (Temperatura_wlot - Temperatura_wylot) < 15.0 THEN
    Sprawnosc_niska := TRUE;
ELSE
    Sprawnosc_niska := FALSE;
END_IF;

// logika czyszczenia obu sekcji
CASE Krok OF
    0: // badanie sprawnosci sekcji i oczekiwanie na odpowiednie cisnienie powietrza
        IF Sprawnosc_niska AND Zgoda_na_przedmuch THEN
            Krok := 1; // start cisnienia pierwszej sekcji
        END_IF;

    1: // przedmuchanie dla pierwszej sekcji
        IF Timer_sekcji.Q THEN
            Krok := 2; // po uplywie czasu przejdz dop drugiej sekcji
        END_IF;

    2: // przedmuchanie drugiej sekcji
        IF Timer_sekcji.Q THEN
            Krok := 3; // Koniec czyszczenia obu sekcji
        END_IF;

    3: // zrestartowanie sekwencji
        Krok := 0;
END_CASE;

// timery - kazda sekcja jest przedmuchiwana przez 8 sekund
Timer_sekcji(IN := (Krok = 1) OR (Krok = 2), PT := T#8s);

// wyjscia
Zawor_sekcji_1 := (Krok = 1) AND Zgoda_na_przedmuch;
Zawor_sekcji_2 := (Krok = 2) AND Zgoda_na_przedmuch;

(* ---- Sterownik_dozownika_karuzelowego.st ---- *)
VAR
    Start_linii          : BOOL;  // przycisk NO uruchamiajacy cyklu linii
    Czujnik_pozycji      : BOOL;  // fotokomorka wykrywajaca opakowanie w gniezdzie dozującym
    Krancowka_indeksu    : BOOL;  // czujnik potwierdzajacy pelny obrot karuzeli o jeden krok

    Timer_dozowania      : TON;   // timer odliczajacy czas otwarcia zaworu do nalewania
    Krok                 : INT;   // krok sekwencji

    Naped_karuzeli       : BOOL;  // silnik obracajacy tarcze
    Zawor_dozujacy       : BOOL;  // elektrozawor nalewajacy
END_VAR

CASE Krok OF
    0: // gotowosc linii - oczekiwanie na start linii
        IF Start_linii THEN
            Krok := 1; // uruchomienie obracania karuzeli
        END_IF;

    1: // obrot karuzeli poszukujac wolnego gniazda
        IF Czujnik_pozycji THEN
            Krok := 2; // Wykryto opakowanie na stanowisku -> zatrzymaj i dozuj
        ELSIF NOT Start_linii THEN
            Krok := 0; // wylaczenie linii
        END_IF;

    2: // nalewanie produktu do opakowania
        IF Timer_dozowania.Q THEN
            Krok := 3; // koniec dozowania, przejdz do stabilizacji
        END_IF;

    3: // czsaowa zwloka po zamknieciu zaworu
        IF Krancowka_indeksu OR Start_linii THEN
            Krok := 1; // kontynuacja obracania i szukanie opakowania
        ELSE
            Krok := 0;
        END_IF;
END_CASE;

// timery
Timer_dozowania(IN := (Krok = 2), PT := T#3500ms);  // czas pelnego otwarcia zaworu dozujacego odmierzajacego dawke

// sterowanie wyjsciami
Naped_karuzeli := (Krok = 1); // silnik kreci sie tylko w kroku 1
Zawor_dozujacy := (Krok = 2); // zawor otwiera sie tylko w kroku 2

(* ---- Sterownik_granulatora_tworzyw.st ---- *)
VAR
    Prad_silnika_glownego : REAL;  // czujnik analogowy odczytujacy prad silnika nozy sprawdzajacy jak ciezko ma silnik (czy noz nie utknal i nie zaklinowal komory)
    Czujnik_temperatury  : REAL;  // czujnik analogowy pomiaru temperatury lozysk - wysoka temperatura = potencjalnie tepe ostrza lub brak smaru
    Przycisk_stop_awaria : BOOL;  // grzyb bezpieczenstwa

    Timer_cofania        : TON;   // timer czasu trwania cofania podajnika
    Krok                 : INT;   // krok sekwencji
    Przeciazenie_nozy    : BOOL;  // bit pamieci zablokowania ostrzy
END_VAR

// powyzej 110 A = zakleszczenie materialu
IF Prad_silnika_glownego > 110.0 THEN
    Przeciazenie_nozy := TRUE;
ELSE
    Przeciazenie_nozy := FALSE;
END_IF;

CASE Krok OF
    0: // maszyna zatrzymana - monitorowanie braku awarii i gotowosci do startu
        IF NOT Przycisk_stop_awaria AND Czujnik_temperatury < 85.0 THEN
            Krok := 1;
        END_IF;

    1: // praca nozy tnących - rozpedzanie kola zamachowego
        Krok := 2; // Po rozruchu przejdz do normalnego podawania

    2: // standardowa praca - podajnik tloczy plastik do komory nozowej
        IF Przycisk_stop_awaria THEN
            Krok := 0; // natychmiastowe zatrzymanie systemu
        ELSIF Przeciazenie_nozy THEN
            Krok := 3; // blokada ostrzy - przejdz do procedury powrotu nozy
        END_IF;

    3: // bezpieczne cofanie podajnika (procedura oczyszczania)
        IF Timer_cofania.Q THEN
            Krok := 2; // powrot do normalnego zasypu po oczyszczeniu
        ELSIF Przycisk_stop_awaria THEN
            Krok := 0;
        END_IF;
END_CASE;

// timer
Timer_cofania(IN := (Krok = 3), PT := T#5s);

(* ---- Sterownik_miksera.st ---- *)
VAR
    Start_procesu         : BOOL;  // przycisk startu cyklu mieszania
    Czujnik_pelny         : BOOL;  // czujnik wysokiego poziomu w zbiorniku (ciecz osiagnela limit)
    Czujnik_pusty         : BOOL;  // czujnik niskiego poziomu (zbiornik zostal oprozniony)

    Timer_mieszania       : TON;   // timer odliczajacy czas pracy mieszadla
    Etap_procesu          : INT;   // krok sekwencji: 0-stop, 1-dozowanie, 2-mieszanie, 3-spust

    Zawor_skladnik_A      : BOOL;  // cewka otwierajaca zawor pierwszy skladnika A
    Zawor_skladnik_B      : BOOL;  // cewka otwierajaca zawor pierwszy skladnika B
    Silnik_mieszadla      : BOOL;  // silnik mieszajacy skladniki
    Zawor_spustowy        : BOOL;  // zawor podajacy gotowy produkt
END_VAR

CASE Etap_procesu OF
    0: // oczekiwanie na uruchomienie programu
        IF Start_procesu AND Czujnik_pusty THEN
            Etap_procesu := 1; // przejscie do podania skladnikow
        END_IF;

    1: // podawanie skladnikow do zapelnienia zbiornika
        IF Czujnik_pelny THEN
            Etap_procesu := 2; // gdy zbiornnik jest pelen nastepuje mieszanie skladnikow
        END_IF;

    2: // miksowanie skladnikow przez okeslony czas
        IF Timer_mieszania.Q THEN
            Etap_procesu := 3; // gdy czas minal przejscie do odbioru produktu
        END_IF;

    3: // oproznienie zbiornika
        IF Czujnik_pusty THEN
            Etap_procesu := 0; // gdy zbiornik jest pusty powrot do oczekiwania
        END_IF;
END_CASE;

// kontrola czasu
Timer_mieszania(IN := (Etap_procesu = 2), PT := T#10s);

// sterowanie ukladem sekwencyjnym na podstawie kroku ukladu
Zawor_skladnik_A := (Etap_procesu = 1); // Zawór komponentu A otwarty w kroku 1
Zawor_skladnik_B := (Etap_procesu = 1); // Zawór komponentu B otwarty w kroku 1
Silnik_mieszadla := (Etap_procesu = 2); // Silnik mieszadła pracuje wyłącznie w kroku 2
Zawor_spustowy   := (Etap_procesu = 3); // Zawór spustowy otwarty w kroku 3

(* ---- Sterownik_napelniania_duzych_workow.st ---- *)
VAR
    Start_napelniania    : BOOL;  // przycisk monostabilny NO stratujacy napelnianie
    Waga_prog_90         : BOOL;  // czujnik PNP osiagniecia 90 procent objetosci na wadze
    Waga_prog_100        : BOOL;  // czujnik PNP maksymalnej objetosci na wadze
    Worek_zalozony       : BOOL;  // czujnik bezpieczenstwa zalozonego worka

    Timer_odpylania      : TON;   // czas pracy ojazdu worka po dozowaniu
    Krok                 : INT;   // krok sekwencji

    Zawor_gruby          : BOOL;  // glowny zawor duzego przeplywu - szybki zsyp
    Zawor_dokladny       : BOOL;  // zawor dociagajacy wage
    Odciag_pylu          : BOOL;  // wentylator odpylania stanowiska zsypowego
END_VAR

CASE Krok OF
    0: // oczekiwanie na zawieszenie worka i wystartowanie ukladu
        IF Start_napelniania AND Worek_zalozony THEN
            Krok := 1; // rozpoczecie szybkiego zsypu
        END_IF;

    1: // dozowanie dla maksymalnej wydajnosci
        IF NOT Worek_zalozony THEN
            Krok := 0; // awaryjne przerwanie cyklu przy zerwanym worku z uchwytu
        ELSIF Waga_prog_90 THEN
            Krok := 2; // osiagnieto 90% masy -> powoli dosypuj do 100 procent objetosci
        END_IF;

    2: // dozowanie dokladne - zamkniety zawor glowny, sypie tylko zawor precyzyjny
        IF NOT Worek_zalozony THEN
            Krok := 0;
        ELSIF Waga_prog_100 THEN
            Krok := 3; // osiagnieto wage docelowa -> przejdz do odpylania
        END_IF;

    3: // odpylanie strefy zasypu przed odczepieniem kontenera
        IF Timer_odpylania.Q OR NOT Worek_zalozony THEN
            Krok := 0; // zakonczono cykl -> powrot do stanu gotowosci
        END_IF;
END_CASE;

// timery
// Odciag pracuje jeszcze przez 4 sekundy po zamknieciu zaworow, aby usunac zawieszony pyl
Timer_odpylania(IN := (Krok = 3), PT := T#4s);

// wyjscia
Zawor_gruby    := (Krok = 1) AND Worek_zalozony;
Zawor_dokladny := ((Krok = 1) OR (Krok = 2)) AND Worek_zalozony;
Odciag_pylu    := (Krok = 1) OR (Krok = 2) OR (Krok = 3); // prezz cala prace odciaganie pylu

(* ---- Sterownik_napowietrzania_osadnika.st ---- *)
VAR
    Sonda_tlenowa            : REAL;  // czujnik analogowy odczytujacy poziomu tlenu zakres 0-10
    Wymuszenie_czyszczenia   : BOOL;  // przycisk lub sygnal usuwania osadu
    Zgarniacz_krancowka      : BOOL;  // czujnik powrotu do pozycji wyjsciowej zgarniacza

    Timer_czyszczenia        : TON;   // czas pelnego cyklu
    Krok_czyszczenia         : INT;   // krok sekwencji

    Dmuchawa_napowietrzania  : BOOL;  // dmuchawa podajaca powietrze na komore
    Naped_zgarniacza         : BOOL;  // silnik mechanizmu zgarniania
    Pompa_osadu              : BOOL;  // pompa usuwajaca osad
END_VAR

// prawidlowy poziom tlenu 2-3 mg/l
IF Sonda_tlenowa < 2.0 THEN
    Dmuchawa_napowietrzania := TRUE;  // Zbyt malo tlenu -> wlacz dmuchawe
ELSIF Sonda_tlenowa > 3.0 THEN
    Dmuchawa_napowietrzania := FALSE; // Poziom osiagniety -> wylacz dmuchawe (oszczednosc energii)
END_IF;

// logika czyszczenia dna
CASE Krok_czyszczenia OF
    0: // uklad oczekuje na sygnal oczyszczania
        IF Wymuszenie_czyszczenia AND Zgarniacz_krancowka THEN
            Krok_czyszczenia := 1;
        END_IF;

    1: // praca zgarniacza
        IF Timer_czyszczenia.Q THEN
            Krok_czyszczenia := 2; // zgarniacz dojechal do konca -> uruchomic pompe
        END_IF;

    2: // odpompowanie osadu
        IF NOT Wymuszenie_czyszczenia THEN
            Krok_czyszczenia := 3; // cykl zakonczony poprawnie -> powrot mechanizmu
        END_IF;

    3: // powrot zgarniacza do pozycji poczatkowej
        IF Zgarniacz_krancowka THEN
            Krok_czyszczenia := 0; // Ckoniec cyklu - oczekiwanie na nowy cykl
        END_IF;
END_CASE;

// timery - czas jazdy zgarniacza wynosi 45 sekund
Timer_czyszczenia(IN := (Krok_czyszczenia = 1), PT := T#45s);

// sterowanie wyjsciami
Naped_zgarniacza := (Krok_czyszczenia = 1) OR (Krok_czyszczenia = 3);
Pompa_osadu      := (Krok_czyszczenia = 2);

(* ---- Sterownik_neutralizacji_sciekow.st ---- *)
VAR
    Uruchom_proces       : BOOL;  // przycisk NO startu cyklu neutralizacji
    Pomiar_pH            : REAL;  // analogowy odczyt wartosci pH (0.0 - 14.0)
    Zbiornik_pelny       : BOOL;  // czujnik poziomu max potwierdzajacy gotowosc porcji

    Timer_dozowania      : TON;   // timer limitujacy czas pojedynczego wtrysku chemii
    Krok                 : INT;   // krok

    Pompa_kwasu          : BOOL;  // pompa dozujaca korektor pH- (kwas)
    Pompa_zasady         : BOOL;  // pompa dozujaca korektor pH+ (zasada)
    Silnik_mieszadla     : BOOL;  // silnik mieszadla zbiornika reakcyjnego
    Zezwolenie_zrzutu    : BOOL;  // sygnal gotowosci do oproznienia zbiornika
END_VAR

CASE Krok OF
    0: // oczekiwanie na pelny zbiornik i sygnal startu
        IF Uruchom_proces AND Zbiornik_pelny THEN
            Krok := 1;
        END_IF;

    1: // analiza pH cieczy
        IF Pomiar_pH > 8.5 THEN
            Krok := 2; // odczyn zbyt zasadowy -> wymagany kwas
        ELSIF Pomiar_pH < 6.5 THEN
            Krok := 3; // odczyn zbyt kwasny -> wymagana zasada
        ELSIF Pomiar_pH >= 6.5 AND Pomiar_pH <= 8.5 THEN
            Krok := 4; // pH w normie -> przejdz do koncowej homogenizacji i zrzutu
        END_IF;

    2: // dodawanie kwasu (pH w dol)
        IF Timer_dozowania.Q OR NOT Uruchom_proces THEN
            Krok := 1; // strzal chemii i wroc do analizy
        END_IF;

    3: // Dozowanie zasady (korekta pH w gore)
        IF Timer_dozowania.Q OR NOT Uruchom_proces THEN
            Krok := 1; // po strzal chemii wroc do analizy i mieszania
        END_IF;

    4: // ostatnie mieszanie i wystawienie na spust sciekow
        IF NOT Zbiornik_pelny OR NOT Uruchom_proces THEN
            Krok := 0; // zbiornik oprozniony -> koniec cyklu
        END_IF;
END_CASE;

// timery
// impuls dodawania chemii trwa max 3 sekundy aby uniknac przebodzcowania odczynu cieczy w zbiorniku
Timer_dozowania(IN := (Krok = 2) OR (Krok = 3), PT := T#3s);

// mieszadlo pracuje podczas trwania calego procesu korekty pH w zbiorniku
Silnik_mieszadla := (Krok > 0);

// sterowanie wyjsciami
Pompa_kwasu       := (Krok = 2) AND Uruchom_proces;
Pompa_zasady      := (Krok = 3) AND Uruchom_proces;
Zezwolenie_zrzutu := (Krok = 4) AND Zbiornik_pelny;

(* ---- Sterownik_odzysku_ciepla.st ---- *)
VAR
    Temp_oleju_kompresora : REAL;  // pomiar temperatury oleju sprezarki
    Temp_zbiornika_co    : REAL;  // pomiar temperatury w zbiorniku
    Zezwolenie_pracy     : BOOL;  // sygnal potwierdzajacy prace kompresora

    Timer_stabilizacji   : TON;   // timer stabilizujacy prace pompy
    Krok                 : INT;   // krok sekwencji: 0-oczekiwanie, 1-weryfikacja, 2-odzysk aktywny

    Pompa_obiegowa_odzysku: BOOL; // pompa podajaca czynnik przez wymiennik
    Zawor_trojdrogowy    : BOOL;  // zawor przekierowujacy przeplyw
END_VAR

CASE Krok OF
    0: // Oczekiwanie na odpowiednie warunki przy pracujacej sprezarce
        IF Zezwolenie_pracy AND (Temp_oleju_kompresora > 75.0) AND (Temp_zbiornika_co < 60.0) THEN
            Krok := 1; // Przekroczono prog -> przejdz do weryfikacji
        END_IF;

    1: // Weryfikacja stabilnosci - warunki musza sie utrzymac przez okreslony czas
        IF NOT Zezwolenie_pracy OR (Temp_oleju_kompresora < 72.0) OR (Temp_zbiornika_co >= 62.0) THEN
            Krok := 0; // Warunki ulegly pogorszeniu -> powrot do oczekiwania
        ELSIF Timer_stabilizacji.Q THEN
            Krok := 2; // Temperatura stabilna -> aktywacja odzysku ciepla
        END_IF;

    2: // Odzysk energii odpadowej
        IF NOT Zezwolenie_pracy OR (Temp_oleju_kompresora < 68.0) OR (Temp_zbiornika_co >= 65.0) THEN
            Krok := 0; // Osiagnieto limit lub sprezarka stanela -> stop odzysku
        END_IF;
END_CASE;

// timery
// Warunki startu musza byc spelnione nieprzerwanie przez 5 sekund, aby uniknac uderzen hydraulicznych
Timer_stabilizacji(IN := (Krok = 1), PT := T#5s);  // warunek startu musi byc spelniony przez conajmniej 5 sekund

// krok sterowania pompami
Pompa_obiegowa_odzysku := (Krok = 2);
Zawor_trojdrogowy      := (Krok = 2);

(* ---- Sterownik_oswietlenia.st ---- *)
VAR
    Zasilanie_glowne_OK : BOOL;       // status zasilania sieciowego (TRUE = jest napięcie)
    Czujnik_zmierzchu   : BOOL;       // TRUE = jest ciemno na zewnątrz
    Wymuszenie_reczne   : BOOL;       // przycisk testowy na szafie (Styk NO)

    Oswietlenie_ewakuacja : BOOL;    // wyjście na lampy awaryjne
END_VAR

// Logika: Włącz światła awaryjne, jeśli brakuje zasilania głównego
// LUB gdy jest ciemno i operator wciśnie przycisk testowy
Oswietlenie_Ewakuacja := NOT Zasilanie_Glowne_OK OR (Czujnik_Zmierzchu AND Wymuszenie_Reczne);

(* ---- Sterownik_oswietlenia_awaryjnego.st ---- *)
VAR
    Zasilanie_glowne_OK : BOOL;       // status zasilania sieciowego (TRUE = sieciowe OK)
    Czujnik_zmierzchu   : BOOL;       // TRUE = noc / ciemność w strefie
    Wymuszenie_reczne   : BOOL;       // przycisk testowy na elewacji szafy (Styk NO)
    Stabilizacja_sieci  : TON;        // timer opóźniający powrót do normalnego zasilania
    Oswietlenie_ewakuacja : BOOL;     // wyjście lamp awaryjnych
END_VAR

// 1. liczymy czas stabilizacji sieci (np. prąd wraca, ale czekamy 5 sekund czy napięcie jest stabilne)
Stabilizacja_sieci(IN := Zasilanie_glowne_OK, PT := T#5s);

// 2. logika załączenia oświetlenia awaryjnego:
// swiatła świecą jeśli sieć nie jest jeszcze stabilna lub gdy operator wymusi test po zmroku
Oswietlenie_ewakuacja := NOT Stabilizacja_sieci.Q OR (Czujnik_zmierzchu AND Wymuszenie_reczne);

(* ---- Sterownik_oswietlenia_klatki.st ---- *)
VAR
    Przycisk : BOOL;               // Przycisk NO na ścianie
    Czujnik_ruchu : BOOL;          // Detektor obecności
    Fotokomorka_jasno : BOOL;      // Czujnik zmierzchowy (TRUE = dzień)
    Lampa_wyjscie : BOOL;          // Stycznik światła
    Lampa_dimmer : INT;            // Jasność 0-100%

    Timer_swiatla : TON;           // Czas świecenia w trybie Auto
    Timer_przycisku : TON;         // Wykrywanie wcisniecia
    Tryb_reczny : BOOL;            // Zmienna trybu stałego
    Blokada_Zmiany : BOOL;         // Zmienna pomocnicza
END_VAR

// 1. Wykrywanie dlugiego przycisniecia (> 3s)
Timer_przycisku(IN := Przycisk, PT := T#3S);

IF Timer_przycisku.Q AND NOT Blokada_Zmiany THEN
    Tryb_reczny := NOT Tryb_reczny;
    Blokada_Zmiany := TRUE;
END_IF;

IF NOT Przycisk THEN
    Blokada_Zmiany := FALSE;
END_IF;

// 2. Logika automatyczna
Timer_swiatla(
    IN := (Czujnik_ruchu OR Przycisk) AND NOT Fotokomorka_jasno AND NOT Tryb_reczny,
    PT := T#30S
);

// 3. Sterowanie Wyjściem
IF Tryb_reczny THEN
    Lampa_wyjscie := TRUE;
    Lampa_dimmer := 100;

ELSIF Timer_swiatla.IN AND NOT Timer_swiatla.Q THEN
    Lampa_wyjscie := TRUE;

    // Funkcja ostrzegawcza (Pre-warning)
    IF Timer_swiatla.ET > T#25S THEN
        Lampa_dimmer := 30;
    ELSE
        Lampa_dimmer := 100;
    END_IF;

ELSE
    Lampa_wyjscie := FALSE;
    Lampa_dimmer := 0;
END_IF;

(* ---- Sterownik_oświetlenia_hali.st ---- *)
VAR
    Sygnal_przetwornika   : INT;    // sygnal z czujnika
    Luks                  : REAL;   // przeliczona wartosc natezenia swiatla
    Czujnik_ruchu         : BOOL;   // wejscie czujnika ruchu
    Godzina_system        : INT;    // daktyczna godzina
    Swiatlo_hala          : BOOL;   // wyjscie na swiatlo na hali
    Opoznienie_ruch       : TOF;    // blok czasowy
END_VAR

// skalowanie - 0 - 1000 luks
Luks := (INT_TO_REAL(NatezenieSwiatla) / 27648.0) * 1000.0;

// opoznione wylaczenie swiatla(15 min)
Timeropoznienia(IN := CzujnikRuchu, PT := T#15M);

// logika sterowania
IF Godzina >= 7 AND Godzina <= 16 THEN  // jesli godzina jest miedzy 7 a 16
    // W godzinach pracy sterowanie tylko jasnoscia
    IF Luks < PrógZalaczenia THEN  // zapal jestli swiatlo ponizej progu
        WyjscieSwiatlo := TRUE;
    ELSIF Luks > (PrógZalaczenia + Histereza) THEN  // jesli swiatlo ponizej progu, to wylacz
        WyjscieSwiatlo := FALSE;
    END_IF;
ELSE
    // poza powyzszymi godzinami, swiatlo dziala tylko gdy jest ciemno
    IF Luks < PrógZalaczenia AND TimerOpoznienia.Q THEN
        WyjscieSwiatlo := TRUE;
    ELSE
        WyjscieSwiatlo := FALSE;
    END_IF;
END_IF;

(* ---- Sterownik_paletyzacji_kartonów.st ---- *)
VAR
    Czujnik_kartonu      : BOOL;  // czujnik optyczny wykrywajacy kartony na koncu tasmy
    Paleta_obecna        : BOOL;  // czujnik obecnosci palety w strefie zaladunku
    Przycisk_reset       : BOOL;  // reset licznika po zabraniu pelnej palety

    Licznik_kartonow     : INT;   // aktualna liczba kartonow na aktualnej warstwie
    Krok                 : INT;   // krok sekwencji

    Tasma_doprowadzajaca : BOOL;  // silnik tasmy podajacej kartony
    Silownik_popychacza  : BOOL;  // pneumatyczny popychacz formujacy warstwe
    Sygnalizacja_pelna   : BOOL;  // lampka informacyjna dla operatora wozka widlowego
END_VAR

CASE Krok OF
    0: // oczekiwanie na podstawienie pustej palety przez obecnego operatora
        Licznik_kartonow := 0;
        IF Paleta_obecna THEN
            Krok := 1; // Paleta wykryta, uruchom linie podawania
        END_IF;

    1: // zbieranie kartonow aby uformowac pelna warstwe
        IF Licznik_kartonow >= 10 THEN
            Krok := 2; // Zebrano warstwe,  zatrzymaj tasme i zepchnij gotowa palete
        END_IF;

    2: // zepchniecie calej warstwy na palete - po zepchnieciu powrot silownika i wykrycie nowej palety
        IF Licznik_kartonow >= 40 THEN
            Krok := 3; // paleta zapelniona
        ELSE
            Krok := 1; // Wroc do zbierania kolejnej warstwy
        END_IF;

    3: // Strefa zapelniona - oczekiwanie na odbior palety i reset ukladu
        IF Przycisk_reset AND NOT Paleta_obecna THEN
            Krok := 0; // Paleta zabrana, powrot do 0 kroku
        END_IF;
END_CASE;

// sterowanie wyjsciami
Tasma_doprowadzajaca := (Krok = 1) AND Paleta_obecna;
Silownik_popychacza  := (Krok = 2);
Sygnalizacja_pelna   := (Krok = 3);

(* ---- Sterownik_pieca_przemyslowego.st ---- *)
VAR
    Przycisk_start      : BOOL;       // przycisk START procesu (Styk NO)
    Przycisk_stop       : BOOL;       // przycisk STOP NC
    Czujnik_drzwi       : BOOL;       // czujnik otwarcia drzwi (TRUE = Otwarte)
    Temp_RAW            : INT;        // surowy sygnał z karty PT100 (0 - 27648)
    Grzalka             : BOOL;       // stycznik załączający grzałki oporowe
    Wentylator_obiegowy : BOOL;       // stymulacja ruchu powietrza w komorze
    Koniec_procesu      : BOOL;       // lampa sygnalizacyjna na panelu
    Temperatura_aktualna : REAL;      // przeliczona temperatura w °C
    Proces_aktywny      : BOOL;       // flaga informująca, że piec pracuje
    Temperatura_osiagnieta : BOOL;    // flaga zezwolenia na odliczanie czasu
    Timer_pieczenia     : TON;        // zegar liczacy czas trwania procesu
END_VAR

// skalowanie na wartosc w Celcjusza
Temperatura_aktualna := (INT_TO_REAL(Temp_RAW) / 27648.0) * 250.0;

// start/stop procesu
IF Przycisk_Start AND NOT Czujnik_Drzwi AND NOT Przycisk_Stop THEN
    Proces_Aktywny := TRUE;
    Koniec_Procesu := FALSE;
ELSIF Przycisk_Stop OR Timer_Pieczenia.Q THEN
    Proces_Aktywny := FALSE; // wyłączenie procesu przy STOP lub po upływie czasu
END_IF;

// grzałka i wentylator mogą pracować tylko przy aktywnym procesie i zamkniętych drzwiach
IF Proces_Aktywny AND NOT Czujnik_Drzwi THEN
    Wentylator_Obiegowy := TRUE; // termoobieg działa zawsze, gdy piec pracuje

    IF Temperatura_aktualna < 178.0 THEN
        Grzalka := TRUE;
    ELSIF Temperatura_aktualna > 182.0 THEN
        Grzalka := FALSE;
    END_IF;

    // rozpoczynanie odliczania czasu gdy piec sie nagrzeje do 180 stopni
    IF Temperatura_aktualna >= 180.0 THEN
        Temperatura_osiagnieta := TRUE;
    END_IF;

ELSE
    // otwarte drzwi lub wylaczony proces wylaczaja grzanie i wentylacje
    Grzalka := FALSE;
    Wentylator_obiegowy := FALSE;
END_IF;

// timer rusza gdy osiagnelismy zadana temperature, otwarcie drzwizatrzymuje liczenie
Timer_pieczenia(IN := (Proces_aktywny AND Temperatura_osiagnieta AND NOT Czujnik_drzwi),
                PT := T#10m);

// Po odliczeniu czasu zapal lampę końca i zresetuj flagę temperatury
IF Timer_pieczenia.Q THEN
    Koniec_procesu := TRUE;
    Temperatura_osiagnieta := FALSE;
END_IF;

(* ---- Sterownik_prasy_belujacej.st ---- *)
VAR
    Start_automatu       : BOOL;  // przycisk wlaczenia trybu automatycznego prasy
    Fotokomorka_zasypu   : BOOL;  // wykrycie odpadow w komorze zasypowej
    Czujnik_cisnienia    : BOOL;  // czujnik osiagniecia max nacisku prasowania (bela gotowa)
    Krancowka_powrotu    : BOOL;  // czujnik potwierdzajacy pelne cofniecie plyty prasujacej

    Timer_zasypu         : TON;   // timer filtrujacy stala obecnosc materialu przed startem prasy
    Krok                 : INT;   // krok sekwencji: 0-idle, 2-prasowanie, 3-powrot

    Ruch_prasowania      : BOOL;  // zawor wysuwu silownika - zgniatanie
    Ruch_powrotny        : BOOL;  // zawor wsuwu silownika - cofniecie plyty
    Licznik_bel          : CTU;   // licznik sprasowanych bel odpadu
END_VAR

// Sekwencja
CASE Krok OF
    0: // Oczekiwanie na zsyp komory
        IF Start_automatu AND Timer_zasypu.Q AND Krancowka_powrotu THEN
            Krok := 2; // Komora pelna, plyta u gory -> start prasowania
        END_IF;

    2: // Ruch plyty prasujacej w dol - zgniatanie odpadow
        IF Czujnik_cisnienia THEN
            Krok := 3; // Osiagnieto maksymalny zgniot -> przejscie do cofania
        END_IF;

    3: // Powrot plyty prasujacej do samej gory
        IF Krancowka_powrotu THEN
            Krok := 0; // Plyta wrocila bazowo - powrot do oczekiwania
        END_IF;
END_CASE;

// Opoznienie startu - material musi zaslonic fotokomorke przez 3 sekundy aby prasa nie ruszyla na pusto
Timer_zasypu(IN := Fotokomorka_zasypu, PT := T#3s);

// Kontrola wyjsc
Ruch_prasowania := (Krok = 2);
Ruch_powrotny   := (Krok = 3);

// Prowadzenie statystyki
// Licznik zwieksza wartosc na zboczu narastajacym po zwiekszeniu cisnienia
Licznik_bel(CU := Czujnik_cisnienia, R := NOT Start_automatu);

(* ---- Sterownik_prasy_filtracyjnej.st ---- *)
VAR
    Start_cyklu          : BOOL;  // przycisk NO uruchamiajadcyautomatyczne odwadnianie
    Cisnienie_szlamu     : REAL;  // czujnik analogowy odczytujacy cisnienie tloczenia
    Prasa_zamknieta      : BOOL;  // czujnik krancowy pelnego docisku plyt filtrujacych

    Timer_odwadniania    : TON;   // timer liczacy czas fazy tloczenia osadu
    Krok                 : INT;   // krok sekwencji

    Zgoda_pompy          : BOOL;  // pamiec zezwolenia na prace pompy zasilajacej prasowe komory
    Zawor_zasilajacy     : BOOL;  // zawor podawania osadu do prasy
    Silownik_docisku     : BOOL;  // agregat dociskajacy plyty prasy
END_VAR

// Jesli cisnienie przekroczy 12 bar to odcina pompe dla ochrony plyt
IF Cisnienie_szlamu > 12.0 THEN
    Zgoda_pompy := FALSE;
ELSE
    Zgoda_pompy := TRUE;
END_IF;

CASE Krok OF
    0: // oczekiwanie na start
        IF Start_cyklu THEN
            Krok := 1; // Rozpocznij mechaniczne zamykanie komor prasy
        END_IF;

    1: // docisk plyt do stacji roboczej
        IF Prasa_zamknieta THEN
            Krok := 2; // gdy plyty sa zabezpieczone i szaczelne to rozpoczecie tloczenia szlamu
        END_IF;

    2: // filtracja i wciskanie wody pod cisnieniem
        IF Timer_odwadniania.Q OR NOT Zgoda_pompy THEN
            Krok := 3; // Czas filtration-loop minal lub cisnienie graniczne -> koniec fazy
        END_IF;

    3: // odpuszczenie silownika i przejscie do stanu gotowosci
        IF NOT Prasa_zamknieta THEN
            Krok := 0; // prasa jest otwarta a suchy osad zsypany
        END_IF;
END_CASE;

// timery - czas tloczenia i nawadniania trwa 60 sekund
Timer_odwadniania(IN := (Krok = 2) AND Zgoda_pompy, PT := T#60s);

// sterowanie wyjsciami
Silownik_docisku := (Krok = 1) OR (Krok = 2); // trzymanie cisnienia przez caly czas filtracji
Zawor_zasilajacy := (Krok = 2) AND Zgoda_pompy AND Prasa_zamknieta;
